	stManualModeParameter[_Chan].stChannelParameter.stManualOption.bTrafoActive := _MachineMode[_Chan].ManualMode.stManualOption.bTrafoActive;
	stManualModeParameter[_Chan].stChannelParameter.stManualOption.bEcsActive := _MachineMode[_Chan].ManualMode.stManualOption.bEcsActive;
	stManualModeParameter[_Chan].stChannelParameter.stManualOption.eZeroOffset := _MachineMode[_Chan].ManualMode.stManualOption.eZeroOffset;					

	_ManualModeJog:=(_MachineMode[_SelectedChannel].ManualMode.nManualTyp=2) AND _Channel[_SelectedChannel].stCmdModesStates.stModes.Manual;
	_ManualModeInc:=(_MachineMode[_SelectedChannel].ManualMode.nManualTyp=3) AND _Channel[_SelectedChannel].stCmdModesStates.stModes.Manual;
	
	stManualModeParameter[_Chan].stAxisParameter.stControlUnit[0].nLogAxisNr := _MachineMode[_Chan].ManualMode.nLogAxisNumber;   (* Log. Achs Nummer *)
	IF stManualModeParameter[_Chan].stAxisParameter.stControlUnit[0].nLogAxisNr = 0 THEN
		stManualModeParameter[_Chan].stAxisParameter.stControlUnit[0].nLogAxisNr := gpCh[_Chan]^.bahn_state.coord_r[0].log_achs_nr_r;
		_MachineMode[_Chan].ManualMode.nLogAxisNumber := gpCh[_Chan]^.bahn_state.coord_r[0].log_achs_nr_r;
	END_IF
	stManualModeParameter[_Chan].stAxisParameter.stControlUnit[0].nSpeed := LREAL_TO_UDINT(_MachineMode[_Chan].ManualMode.nSpeed * (100000/60));//um/min >> mm/sec
	stManualModeControlElements[_Chan].stControlKeys[0].bKeyNeg := _MachineMode[_Chan].ManualMode.bKeyNeg;
	stManualModeControlElements[_Chan].stControlKeys[0].bKeyPos := _MachineMode[_Chan].ManualMode.bKeyPos;
	stManualModeControlElements[_Chan].stControlKeys[0].bKeyRapid := _MachineMode[_Chan].ManualMode.bKeyRapid;
	
	//Handwheel
	IF _Handwheel.xAxisSelect THEN
		_MachineMode[_Chan].ManualMode.nLogAxisNumber := INT_TO_UINT(_Axis[0].nLogAxisNo);
	ELSIF _Handwheel.yAxisSelect THEN
		_MachineMode[_Chan].ManualMode.nLogAxisNumber := INT_TO_UINT(_Axis[1].nLogAxisNo);
	ELSIF _Handwheel.zAxisSelect THEN
		_MachineMode[_Chan].ManualMode.nLogAxisNumber := INT_TO_UINT(_Axis[2].nLogAxisNo);
	ELSIF _Handwheel.aAxisSelect THEN
		_MachineMode[_Chan].ManualMode.nLogAxisNumber := INT_TO_UINT(_Axis[3].nLogAxisNo);
	ELSIF _Handwheel.cAxisSelect THEN
		_MachineMode[_Chan].ManualMode.nLogAxisNumber := INT_TO_UINT(_Axis[4].nLogAxisNo);
	ELSIF _MachineMode[_Chan].ManualMode.nManualTyp = 1 THEN
		_MachineMode[_Chan].ManualMode.nManualTyp := 0;			
	END_IF
	
	IF _Handwheel.x10Resolution THEN
		_MachineMode[_Chan].ManualMode.nHwResolution := 10;
	ELSIF _Handwheel.x100Resolution THEN
		_MachineMode[_Chan].ManualMode.nHwResolution := 100;
	ELSE
		_MachineMode[_Chan].ManualMode.nHwResolution := 1;
	END_IF
		
	stManualModeParameter[_Chan].stChannelParameter.nHandwheelResolution := UDINT_TO_DINT(_MachineMode[_Chan].ManualMode.nHwResolution)* LREAL_TO_DINT(10000);
	_fbUintUdint[_Chan](ninSmall := _Handwheel.Handwheel, nBig := _HandWheelBig);
	stManualModeControlElements[_Chan].nHandwheelinc[0] :=  UDINT_TO_DINT(_HandWheelBig);
	IF _HandWheelBig > 214748364 OR _HandWheelBig = 0 THEN
		_MachineMode[_Chan].ManualMode.nLogAxisNumber := 0;
		_HandWheelBig := 107374182;
	END_IF
END_IF
END_METHOD

METHOD PRIVATE M_Selections
VAR_INPUT
	{attribute 'tc_no_symbol'}
	_Chan					 : INT;
END_VAR
VAR_INST
END_VAR
//Reset
	_MachineMode[_Chan].Reset := Control.Inputs.AlarmAck.Enabled OR Control.Inputs.Reset.Enabled;

//Energize
	_R_Trig[7](CLK:=Energize); 
	IF _R_Trig[7].Q THEN 
		_AutoEn:= TRUE; 
	END_IF
	
	_R_trig[6](CLK:= NOT Energize); 
	IF _R_Trig[6].Q THEN 
		_AutoEn:= FALSE; 
	END_IF

//Stop
	_R_Trig[8](CLK:=Control.PackMLState.Stopping OR Control.PackMLState.Holding);
	_MachineMode[_SelectedChannel].Stop := _R_Trig[8].Q;

//Start
	_R_Trig[9](CLK:= (Control.PackMLState.Starting OR Control.PackMLState.Execute) AND _AxisEnabled);
	_MachineMode[_SelectedChannel].Start := _R_Trig[9].Q;
	
//Standby Mode
	_StandbyMode.Interlock := Control.PackMLState.Execute  OR (_StandbyMode.Enabled AND _MachineMode[_Chan].Mode <> E_CNC_Mode.STANDBY_MODE);
	IF _StandbyMode.Interlock THEN 
		_StandbyMode.Messages := 'CNC Machine Must not be Executing for Standby Mode'; 
	END_IF;
	
	_StandbyMode.Select := (_StandbyMode.Select) AND NOT _StandbyMode.Interlock;
	IF NOT _StandbyMode.Select AND NOT _StandbyMode.Interlock THEN 
		_StandbyMode.Messages := 'CNC Ready for Standby Mode'; 
	END_IF;
	
	_StandbyMode.Queued := _StandbyMode.Select;
	IF _StandbyMode.Queued AND NOT _StandbyMode.Enabled THEN 
		_StandbyMode.Messages := 'CNC Standby Mode Selection Queued'; 
	END_IF;
	
	_R_Trig[10](CLK:= _StandbyMode.Queued); 
	IF _R_Trig[10].Q THEN 
		_MachineMode[_Chan].Standby := TRUE;
	END_IF;
	
	_StandbyMode.Enabled := _StandbyMode.Queued AND _MachineMode[_Chan].Mode = E_CNC_Mode.STANDBY_MODE;
	IF _StandbyMode.Enabled THEN 
		_StandbyMode.Messages := 'CNC Standby Mode Enabled'; 
	END_IF;

//Automatic Mode Selection
	_AutomaticMode.Interlock := Control.PackMLState.Execute AND NOT _AutomaticMode.Enabled OR (_AutomaticMode.Enabled AND _MachineMode[_Chan].Mode <> E_CNC_Mode.AUTOMATIC_MODE);
	IF _AutomaticMode.Interlock THEN 
		_AutomaticMode.Messages := 'CNC Machine Must not be Executing for Automatic Mode Selection'; 
	END_IF;
	
	_AutomaticMode.Select := _AutomaticMode.Select AND NOT _AutomaticMode.Interlock;
	IF NOT _AutomaticMode.Select AND NOT _AutomaticMode.Interlock THEN
 		_AutomaticMode.Messages := 'CNC Ready for Automatic Mode'; 
	END_IF;
	
	_AutomaticMode.Queued := _AutomaticMode.Select;
	IF _AutomaticMode.Queued AND NOT _AutomaticMode.Enabled THEN 
		_AutomaticMode.Messages := 'CNC Automatic Mode Selection Queued'; 
	END_IF;
	
	_R_Trig[11](CLK:= _AutomaticMode.Queued);
	IF _R_Trig[11].Q THEN 
		_MachineMode[_Chan].Automatic := TRUE;
	END_IF;
	
	_AutomaticMode.Enabled := _AutomaticMode.Queued AND _MachineMode[_Chan].Mode = E_CNC_Mode.AUTOMATIC_MODE;
	IF _AutomaticMode.Enabled THEN 
		_AutomaticMode.Messages := 'CNC Automatic Mode Enabled'; 
	END_IF;

//3 MDI Mode Selection
	_MDIMode.Interlock := Control.PackMLState.Execute AND NOT _MDIMode.Enabled  OR (_MDIMode.Enabled AND _MachineMode[_Chan].Mode <> E_CNC_Mode.MDI_MODE);
	IF _MDIMode.Interlock THEN 
		_MDIMode.Messages := 'CNC Machine Must not be Executing for MDI Mode Selection'; 
	END_IF;
	
	_MDIMode.Select := _MDIMode.Select AND NOT _MDIMode.Interlock;
	IF NOT _MDIMode.Select AND NOT _MDIMode.Interlock THEN 
		_MDIMode.Messages := 'CNC Ready for MDI Mode'; 
	END_IF;
	
	_MDIMode.Queued := _MDIMode.Select;
	IF _MDIMode.Queued AND NOT _MDIMode.Enabled THEN 
		_MDIMode.Messages := 'CNC MDI Mode Selection Queued'; 
	END_IF;
	
	_R_Trig[12](CLK:= _MDIMode.Queued); 
	IF _R_Trig[12].Q THEN 
		_MachineMode[_Chan].MDI:= TRUE;
	END_IF;

	_MDIMode.Enabled := _MDIMode.Queued AND _MachineMode[_Chan].Mode = E_CNC_Mode.MDI_MODE;
	IF _MDIMode.Enabled THEN 
		_MDIMode.Messages := 'CNC MDI Mode Enabled'; 
	END_IF;

//Manual Mode Selection
	_ManualMode.Interlock := (NOT control.PackMLState.Stopped AND NOT control.PackMLState.Idle)OR (_ManualMode.Enabled AND ((_MachineMode[_Chan].Mode <> E_CNC_Mode.MANUAL_MODE)OR _R_Trig[15].Q));
	IF _ManualMode.Interlock THEN 
		_ManualMode.Messages := 'CNC Must be in a Stopped or Idle State for Manual Mode'; 
	END_IF;	_R_Trig[13](CLK:= _ManualMode.Queued);
	
	_ManualMode.Select := _ManualMode.Select AND NOT _ManualMode.Interlock;
	IF NOT _ManualMode.Select AND NOT _ManualMode.Interlock THEN 
		_ManualMode.Messages := 'CNC Ready for Manual Mode'; 
	END_IF;
	
	_ManualMode.Queued := _ManualMode.Select;
	IF _ManualMode.Queued AND NOT _ManualMode.Enabled THEN 
		_ManualMode.Messages := 'CNC Manual Mode Selection Queued'; 
	END_IF;

	IF _R_Trig[13].Q THEN 
		_MachineMode[_Chan].ManualMode.nManualTyp := 2;  _MachineMode[_Chan].Manual := TRUE; 
	END_IF;
	
	_ManualMode.Enabled := _ManualMode.Queued AND (_MachineMode[_Chan].ManualMode.nManualTyp<>1) AND _MachineMode[_Chan].Mode = E_CNC_Mode.MANUAL_MODE;
	IF _ManualMode.Enabled THEN 
		_ManualMode.Messages := 'CNC Manual Mode Enabled';
	END_IF;
	
//5 Reference Mode Selection
	_ReferenceMode.Interlock := NOT Control.PackMLState.Resetting OR (_ReferenceMode.Enabled AND _MachineMode[_Chan].Mode <> E_CNC_Mode.REFERENCE_MODE);
	IF _ReferenceMode.Interlock THEN 
		_ReferenceMode.Messages := 'CNC Must be in a Stopped or Resseting State for Reference Mode'; 
	END_IF;
	
	_ReferenceMode.Select := (_ReferenceMode.Select OR _AutoHome OR _ManHome.Enabled) AND NOT _ReferenceMode.Interlock;
	IF NOT _ReferenceMode.Select AND NOT _ReferenceMode.Interlock THEN 
		_ReferenceMode.Messages := 'CNC Ready for Reference Mode'; 
	END_IF;

	_ReferenceMode.Queued := _ReferenceMode.Select;
	IF _ReferenceMode.Queued AND NOT _ReferenceMode.Enabled THEN 
		_ReferenceMode.Messages := 'CNC Reference Mode Selection Queued'; 
	END_IF;

	_ReferenceMode.Enabled := _ReferenceMode.Queued;
	IF _ReferenceMode.Enabled THEN 
		_ReferenceMode.Messages := 'CNC Reference Mode Enabled';
	END_IF;
	
//Handwheel Mode Selected
	_HandwheelMode.Interlock := (NOT control.PackMLState.Stopped AND NOT control.PackMLState.Idle) OR (_HandwheelMode.Enabled AND ((_MachineMode[_Chan].Mode <> E_CNC_Mode.MANUAL_MODE)OR _R_Trig[13].Q));
	IF _HandwheelMode.Interlock THEN 
		_HandwheelMode.Messages := 'CNC Must be in a Stopped or Idle State for Handwheel Mode'; 
	END_IF;

	_HandwheelMode.Select := (_Handwheel.xAxisSelect OR _Handwheel.yAxisSelect OR _Handwheel.zAxisSelect OR _Handwheel.cAxisSelect OR _Handwheel.aAxisSelect) AND NOT _HandwheelMode.Interlock;
	IF NOT _HandwheelMode.Select AND NOT _HandwheelMode.Interlock THEN 
		_HandwheelMode.Messages := 'CNC Ready for Handwheel Mode'; 
	END_IF;

	_HandwheelMode.Queued := _HandwheelMode.Select;
	IF _HandwheelMode.Queued AND NOT _HandwheelMode.Enabled THEN 
		_HandwheelMode.Messages := 'CNC Handwheel Mode Selection Queued'; 
	END_IF;

	_R_Trig[15](CLK:= _HandwheelMode.Queued);
	IF _R_Trig[15].Q THEN 
		_MachineMode[_Chan].ManualMode.nManualTyp := 1; _MachineMode[_Chan].Manual := TRUE; 
	END_IF;

	_HandwheelMode.Enabled := _HandwheelMode.Queued AND (_MachineMode[_Chan].ManualMode.nManualTyp=1) AND _MachineMode[_Chan].Mode = E_CNC_Mode.MANUAL_MODE;
	IF _HandwheelMode.Enabled THEN 
		_HandwheelMode.Messages := 'CNC Handwheel Mode Enabled'; 
	END_IF;

//Manual Home Selection
	_R_Trig[16](CLK:= _Homed);	
	_ManHome.Interlock := (NOT control.PackMLState.Stopped AND NOT control.PackMLState.Resetting) OR _R_Trig[16].Q;
	IF _ManHome.Interlock THEN 
		_ManHome.Messages := 'CNC Must be in a Stopped State for Manual Homing'; 
	END_IF;
	
	_ManHome.Select := _ManHome.Select AND NOT _ManHome.Interlock;
	IF NOT _ManHome.Select AND NOT _ManHome.Interlock THEN 
		_ManHome.Messages := 'CNC Ready for Selected Axis to be Homed'; 
	END_IF;
	
	_ManHome.Queued := _ManHome.Select;
	IF _ManHome.Queued AND NOT _ManHome.Enabled THEN 
		_ManHome.Messages := 'CNC Waiting for Machine to be put into Resetting'; 
	END_IF;
	
	_ManHome.Enabled := _ManHome.Queued AND Control.PackMLState.Resetting;
	IF _ManHome.Enabled THEN 
		_ManHome.Messages := 'CNC Axis Manual Home Enabled'; 
	END_IF;

//Spindle Warmup
	_SpindleWarmup.Interlock := Spindle.Warm OR (NOT A1_Control.PackMLState.Idle AND NOT A1_Control.PackMLState.Starting AND NOT A1_Control.PackMLState.Execute AND NOT A1_Control.PackMLState.Completing);
	IF _SpindleWarmup.Interlock THEN 
		_SpindleWarmup.Messages := 'Spindle is Warm or CNC is Not in a Suitable State'; 
	END_IF;
	
	_SpindleWarmup.Select := _SpindleWarmup.Select AND NOT _SpindleWarmup.Interlock;
	IF NOT _SpindleWarmup.Select AND NOT _SpindleWarmup.Interlock THEN 
		_SpindleWarmup.Messages := 'Ready for Spindle Warmup'; 
	END_IF;
	
	_SpindleWarmup.Queued := _SpindleWarmup.Select;
	IF _SpindleWarmup.Queued AND NOT _SpindleWarmup.Enabled THEN 
		_SpindleWarmup.Messages := 'Spindle Warmup is Queued'; 
	END_IF;
	
	_SpindleWarmup.Enabled := _SpindleWarmup.Queued AND Control.PackMLState.Execute;
	IF _SpindleWarmup.Enabled THEN 
		_SpindleWarmup.Messages := 'Spindle Warmup Enabled'; 
	END_IF;
	
//Retract Tool
	_RetractTool.Interlock := NOT A1_Control.PackMLState.Idle AND NOT A1_Control.PackMLState.Starting AND NOT A1_Control.PackMLState.Execute AND NOT A1_Control.PackMLState.Completing;
	IF _RetractTool.Interlock THEN 
		_RetractTool.Messages := 'Machine Not in a Suitable State to Retract Tool'; 
	END_IF;
	
	_RetractTool.Select := (_RetractTool.Select) AND NOT _RetractTool.Interlock;
	IF NOT _RetractTool.Select AND NOT _RetractTool.Interlock THEN 
		_RetractTool.Messages := 'Ready for Tool Retract'; 
	END_IF;
	
	_RetractTool.Queued := _RetractTool.Select;
	IF _RetractTool.Queued AND NOT _RetractTool.Enabled THEN 
		_RetractTool.Messages := 'Retract Tool Selection Queued'; 
	END_IF;
	
	_RetractTool.Enabled := _RetractTool.Queued AND Control.PackMLState.Execute;
	IF _RetractTool.Enabled THEN 
		_RetractTool.Messages := 'Retract Tool Enabled'; 
	END_IF;
END_METHOD

METHOD PRIVATE M_Spindle
VAR_INPUT
	{attribute 'tc_no_symbol'}
	_Chan					 : INT;
END_VAR
VAR_INST
	_Delay							: TON;
	_fbHandleSpindleTechno			: HLI3_HandleSpindleTechno;
	_ton							: ARRAY[0..5] OF TON;
	_Step							: UINT;
	_MaxSpeed						: UINT := 24000;
	_r_trig							: ARRAY[0..2] OF R_TRIG;
END_VAR
_fbHandleSpindleTechno(
	nHliAxisIdx:=0, 
	nHliChannelIdx:=_Chan, 	
	bIsChannelSpecific:= TRUE,	
	nRevolution=>Spindle.ComVelocity,
	nLogAxisNoChannelSpecific:= 96, 
	nPosition=> Spindle.Position, 
	bError=> Spindle.Error, 
	nErrorId=> Spindle.ErrorID, 
	M03:= Spindle.M3, 
	M04:= Spindle.M4, 
	M05:= Spindle.M5, 
	M19:= Spindle.M19);

Spindle.ActVelocity:= _Axis[5].stStatus.fActVelo;

// Spindle warm up control
_ton[0](PT:=T#90M, IN:= Spindle.Warm AND NOT SC2501.RunFeedback);
IF _ton[0].Q THEN
	Spindle.Warm := FALSE;
END_IF

CASE _Step OF
	0: //Idle
	IF _SpindleWarmup.Queued THEN
		_Step := 1;
	END_IF
	
	1: //Change to MDI Mode
	_r_trig[0](CLK := TRUE);
	IF _r_trig[0].Q THEN
		_MachineMode[_Chan].MDI := TRUE;
	END_IF

	_MachineMode[_Chan].MDIString := 'T6$R$NM06$R$NM03 S12000$R$NG04 120$R$NM03 S18000$R$NG04 120$R$NM03 S24000$R$NG04 60$R$NM05$R$NT0$R$NM06$R$NG84$R$NM30';
	IF _MachineMode[_Chan].Mode = E_CNC_Mode.MDI_MODE THEN
		_r_trig[0](CLK := FALSE);
		_Step := 2;
		
	ELSIF NOT _SpindleWarmup.Queued THEN
		_Step := 0;
		_MachineMode[_Chan].MDIString := '';
		_MachineMode[_Chan].Standby := TRUE;
	END_IF
	
	2: //Start
	Control.Inputs.Start.Enabled:= TRUE;
	
	IF _MachineMode[_Chan].State = E_CNC_State.ACTIVE AND _SpindleWarmup.Enabled THEN
		_r_trig[0](CLK := FALSE);
		_Step := 3;
	ELSIF NOT _SpindleWarmup.Queued THEN
		_Step := 0;
		_MachineMode[_Chan].MDIString := '';
		_MachineMode[_Chan].Standby := TRUE;
	END_IF
	
	3: //Complete
	IF _ProgramEnd[_Chan] THEN
		Spindle.Warm := TRUE;
		_SpindleWarmup.Select:= FALSE;
		_MachineMode[_Chan].MDIString := '';
		_Step := 0;
		_MachineMode[_Chan].Standby := TRUE;
	ELSIF NOT _SpindleWarmup.Enabled THEN
		_Step := 0;
		_MachineMode[_Chan].MDIString := '';
		_MachineMode[_Chan].Standby := TRUE;
	END_IF
END_CASE
END_METHOD

METHOD PRIVATE M_ToolHandler
VAR_INPUT
	{attribute 'tc_no_symbol'}
	_Chan					 : INT;
END_VAR
VAR_INST
	_r_trig					: ARRAY[0..5] OF R_TRIG;
	_f_trig					: ARRAY[0..2] OF F_TRIG;
	_Step					: UINT;
END_VAR
_ToolData[0].tool_desc.tool_id.basic := 0;
_ToolData[0].tool_desc.valid := TRUE;

//Transfer Tool Data for Requested Tool from Database
IF _Channel[_Chan].pChannel^.ToolData.bToolRequest THEN
	CASE _Channel[_Chan].pChannel^.ToolData.nToolRequestID OF
	0:
		_Channel[_Chan].pChannel^.ToolData.stActTool := _ToolData[0];	
	1:
		_Channel[_Chan].pChannel^.ToolData.stActTool := _ToolData[1];	
	2:
		_Channel[_Chan].pChannel^.ToolData.stActTool := _ToolData[2];	
	3:
		_Channel[_Chan].pChannel^.ToolData.stActTool := _ToolData[3];	
	4:
		_Channel[_Chan].pChannel^.ToolData.stActTool := _ToolData[4];	
	5:
		_Channel[_Chan].pChannel^.ToolData.stActTool := _ToolData[5];	
	6:
		_Channel[_Chan].pChannel^.ToolData.stActTool := _ToolData[6];	
		
	END_CASE		
END_IF

//Transfer Tool Data from Currently used tool back into Database
IF _Channel[_Chan].pChannel^.ToolData.bOldToolDataExist THEN
	_Channel[_Chan].pChannel^.ToolData.bOldToolDataExist := FALSE;
END_IF

//Reply of request read and processed
IF _Channel[_Chan].pChannel^.ToolData.nToolRequestID = _Channel[_Chan].pChannel^.ToolData.stActTool.tool_desc.tool_id.basic THEN
	_Channel[_Chan].pChannel^.ToolData.bToolRequest := FALSE;
END_IF

//Tool Holder
_r_trig[0](CLK:= _Channel[_Chan].pChannel^.M[7].bState_rw);
IF _r_trig[0].Q THEN
	Spindle.M7:= TRUE;
END_IF

_f_trig[0](CLK:= Spindle.M7);
IF _f_trig[0].Q THEN
	_Channel[_Chan].pChannel^.M[7].bState_rw:= FALSE;
END_IF

_r_trig[1](CLK:= _Channel[_Chan].pChannel^.M[8].bState_rw);
IF _r_trig[1].Q THEN
	Spindle.M8:= TRUE;
END_IF

_f_trig[1](CLK:= Spindle.M8);
IF _f_trig[1].Q THEN
	_Channel[_Chan].pChannel^.M[8].bState_rw:= FALSE;
END_IF

_r_trig[2](CLK:= _Channel[_Chan].pChannel^.M[9].bState_rw);
IF _r_trig[2].Q THEN
	Spindle.M9:= TRUE;
END_IF

_f_trig[2](CLK:= Spindle.M9);
IF _f_trig[2].Q THEN
	_Channel[_Chan].pChannel^.M[9].bState_rw:= FALSE;
END_IF

//Tool Retract
IF NOT _RetractTool.Queued THEN
	_Step:= 0;
END_IF

CASE _Step OF
	0: //Idle
	IF _RetractTool.Queued THEN
		_Step := 1;
	END_IF
	
	1: //Change to MDI Mode
	_r_trig[3](CLK := TRUE);
	IF _r_trig[3].Q THEN
		_MachineMode[_Chan].MDI := TRUE;
	END_IF
	
	_MachineMode[_Chan].MDIString := 'G85$R$NX8000 Y650 Z-135 C90 A-90$R$NM02';
	IF _MachineMode[_Chan].Mode = E_CNC_Mode.MDI_MODE THEN
		_r_trig[3](CLK := FALSE);
		_Step := 2;
	END_IF
	
	2: //Start
	Control.Inputs.Start.Select:= TRUE;
	
	IF _MachineMode[_Chan].State = E_CNC_State.ACTIVE THEN
		_Step := 3;
	END_IF
	
	3: //Complete
	IF _ProgramEnd[_Chan] THEN//_MachineMode[_Chan].State = E_CNC_State.READY THEN
		_Step := 0;
		_MachineMode[_Chan].MDIString := '';
		_RetractTool.Select:= FALSE;
		_MachineMode[_Chan].Standby := TRUE;
	END_IF
END_CASE
END_METHOD

METHOD PRIVATE M_VariableViewer
VAR_INST
	_fbReadCNCVariables 	: FB_ReadCNCVariables;
END_VAR
_fbReadCNCVariables(
	bEnable:= TRUE, 
	nChanIdx:= _SelectedChannel, 
	eVariablesType:= eVariablesType, 
	tIntervall:= T#1S, 	 
	stCNCVariablesViewer_Data:= stCNCVariablesViewer_Data);

_pVE_Chan0:= HLI3_LinkVEChannelStructure(nChanIdx:= 0, bGlobal:= FALSE);

_pVE_Chan0^.ParkPos.X:=  _ParkPositions[0];
_pVE_Chan0^.ParkPos.Y:=  _ParkPositions[1];
_pVE_Chan0^.ParkPos.Z:=  _ParkPositions[2];
_pVE_Chan0^.ParkPos.C:=  _ParkPositions[3];
_pVE_Chan0^.ParkPos.A:=  _ParkPositions[4];
END_METHOD

METHOD PRIVATE M_WarningMonitor
VAR_INPUT
END_VAR
VAR_INST
END_VAR
VAR_INST // added by the converter: edge detectors and wires of the graphical bodies
    _w1 : BOOL;
END_VAR
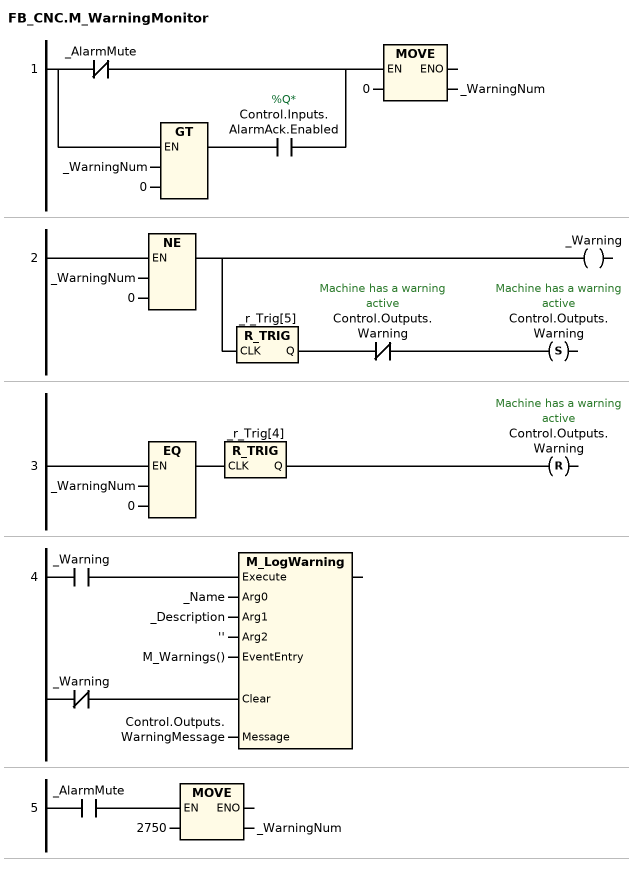
// NETWORK 1
//   Control.Inputs.AlarmAck.Enabled: AT %Q*
IF NOT _AlarmMute OR _WarningNum > 0 AND Control.Inputs.AlarmAck.Enabled THEN _WarningNum := 0; END_IF

// NETWORK 2
//   Control.Outputs.Warning: Machine has a warning active
_w1 := _WarningNum <> 0;
_Warning := _w1;
_r_Trig[5](CLK := _w1); // R_TRIG
Control.Outputs.Warning S= _r_Trig[5].Q AND NOT Control.Outputs.Warning;

// NETWORK 3
//   Control.Outputs.Warning: Machine has a warning active
_r_Trig[4](CLK := _WarningNum = 0); // R_TRIG
Control.Outputs.Warning R= _r_Trig[4].Q;

// NETWORK 4
M_LogWarning(Execute := _Warning, Arg0 := _Name, Arg1 := _Description, Arg2 := '', EventEntry := M_Warnings(), Clear := NOT _Warning, Message := Control.Outputs.WarningMessage);

// NETWORK 5
IF _AlarmMute THEN _WarningNum := 2750; END_IF
END_METHOD

METHOD PRIVATE M_Warnings : TcEventEntry
VAR_INPUT
END_VAR
CASE _WarningNum OF		
	2750: M_Warnings:= TC_Events.TcCnc.W_2750;//Alarm Mute Active						
ELSE
	M_Warnings:=  TC_Events.TcCnc.W_Undefined;
END_CASE
END_METHOD

PROPERTY PUBLIC MachineMode : REFERENCE TO ARRAY[0..3] OF ST_MachineMode;
GET
MachineMode REF= _MachineMode;
END_GET
END_PROPERTY

{attribute 'monitoring' := 'variable'}
PROPERTY PUBLIC Name : String[15]
GET
Name := _Name;
END_GET
SET
_Name := Name;
END_SET
END_PROPERTY

PROPERTY PUBLIC ProgramEnd : REFERENCE TO ARRAY[0..3] OF  BOOL
GET
ProgramEnd REF= _ProgramEnd;
END_GET
END_PROPERTY

PROPERTY PUBLIC ToolData : ARRAY [0..6] OF ST_CNC_TOOL_DATA_EXT
SET
_ToolData:= ToolData;
END_SET
END_PROPERTY

PROPERTY PUBLIC Variables : REFERENCE TO ARRAY[0..9] OF ST_Variable
GET
Variables REF= _Variables;
END_GET
END_PROPERTY

{attribute 'monitoring' := 'variable'}
PROPERTY PUBLIC Warning : Bool
GET
Warning := _Warning;
END_GET
END_PROPERTY

END_FUNCTION_BLOCK

// Objects/FB_CsvLogger_V1_01/FB_CsvLogger
FUNCTION_BLOCK FINAL FB_CsvLogger EXTENDS FB_EventLogger  
VAR_INPUT
	Write					: BOOL;							//Write Log
	HeaderString			: ARRAY[0..9] OF STRING;		//Header Strings
	DataString				: ARRAY[0..9] OF STRING;		//Data Strings
END_VAR                                          	    	
VAR_IN_OUT                                          		
	Control					: ST_System;            		//Machine Control Instance
END_VAR                                             		                                           	
VAR                                                     	
	_Export					: BOOL;							//Export CSV to file destination
	_Fault					: BOOL;	     					//Device Fault
	_SeekPos				: DINT;							//Bytes Logged
	_FaultTimer_ET			: REAL;							//Fault timer elapsed
	_fbCreateDir 			: FB_CreateDir;					//Create File Directory Funciton
	_fbFileOpen				: FB_FileOpen;              	//File Open Function      
	_fbFileClose			: FB_FileClose;             	//File Close Function            
    _fbFileRead             : FB_FileRead;              	//File Read Function 			          
    _fbFileWrite            : FB_FileWrite;             	//File Write Function 	          
	_fbFileDelete  			: FB_FileDelete;            	//File Delete Function           
    _fbFileSeek             : FB_FileSeek;              	//File Seek Function             
	_fbFileTell 			: FB_FileTell;              	//File Tell Function 			          
	_fbFindFileEntry 		: FB_EnumFindFileEntry;     	//File Find File Function 		      
    _hSrcFile               : UINT := 0;					//Temporary file handler
 	_hDestFile              : UINT := 0;					//Export file handler
	_Alarm					: BOOL;							//Device Alarm
	_Warning				: BOOL;							//Device Warning
	_AlarmNum				: DINT;							//Device Alarm Number
	_WarningNum				: DINT;							//Device Warning Number
	_ExtendedErrorCode		: UDINT;						//Extended Error Code
	_R_Trig					: ARRAY[0..9] OF R_TRIG;		//Private Rising Edge Triggers
END_VAR
VAR PERSISTENT
	_Enable					: BOOL;							//Enable CSV logging
	_MaxFileSize			: DINT := 100000;           	//Maximum file size in bytes
	_Name					: STRING[15];					//Name for HMI
	_Description			: STRING[40];					//Description for HMI
	_AlarmMute				: BOOL;							//Alarm Mute
	_FaultTimer_PT			: REAL;							//Fault timer preset time
	_TempFilePath			: STRING:='C:\TwinCAT\3.1\Boot\';//Temporary File Path
	_ExportFilePath			: STRING:='C:\TwinCAT\';		//Export File Path
END_VAR

M_AlarmMonitor();
M_WarningMonitor();
M_Log();

{attribute 'monitoring' := 'variable'}
PROPERTY PUBLIC Alarm : Bool
GET
Alarm := _Alarm;
END_GET
END_PROPERTY

{attribute 'monitoring' := 'variable'}
PROPERTY PUBLIC AlarmMute : BOOL
SET
AlarmMute := _AlarmMute;
END_SET
END_PROPERTY

{attribute 'monitoring' := 'variable'}
PROPERTY PUBLIC Description : String[40]
GET
Description := _Description;
END_GET
SET
_Description := Description;
END_SET
END_PROPERTY

{attribute 'monitoring' := 'variable'}
PROPERTY PUBLIC Enable : BOOL
GET
Enable := _Enable;
END_GET
SET
_Enable := Enable;
END_SET
END_PROPERTY

{attribute 'monitoring' := 'variable'}
PROPERTY PUBLIC Fault : Bool
SET
_Fault := Fault;
END_SET
END_PROPERTY

{attribute 'monitoring' := 'variable'}
PROPERTY PUBLIC FaultTimer_ET : real
GET
FaultTimer_ET := _FaultTimer_ET;
END_GET
END_PROPERTY

{attribute 'monitoring' := 'variable'}
PROPERTY PUBLIC FaultTimer_PT : real
GET
FaultTimer_PT := _FaultTimer_PT;
END_GET
SET
_FaultTimer_PT := FaultTimer_PT;
END_SET
END_PROPERTY

METHOD FB_exit : BOOL
VAR_INPUT
	bInCopyCode : BOOL; // if TRUE, the exit method is called for exiting an instance that is copied afterwards (online change).
END_VAR
IF _hSrcFile <> 0 THEN
	_fbFileClose( bExecute := FALSE );	
	_fbFileClose(sNetId:='', hFile:=_hSrcFile, bExecute:=TRUE, tTimeout:=DEFAULT_ADS_TIMEOUT);
END_IF
END_METHOD

METHOD PRIVATE M_AlarmMonitor
VAR_INPUT
END_VAR
VAR_INST // added by the converter: edge detectors and wires of the graphical bodies
    _w1, _w2, _w3, _w4, _w5, _w6, _w7 : BOOL;
    _rt1, _rt2, _rt3, _rt4, _rt5, _rt6, _rt7, _rt8, _rt9, _rt10 : R_TRIG;
END_VAR
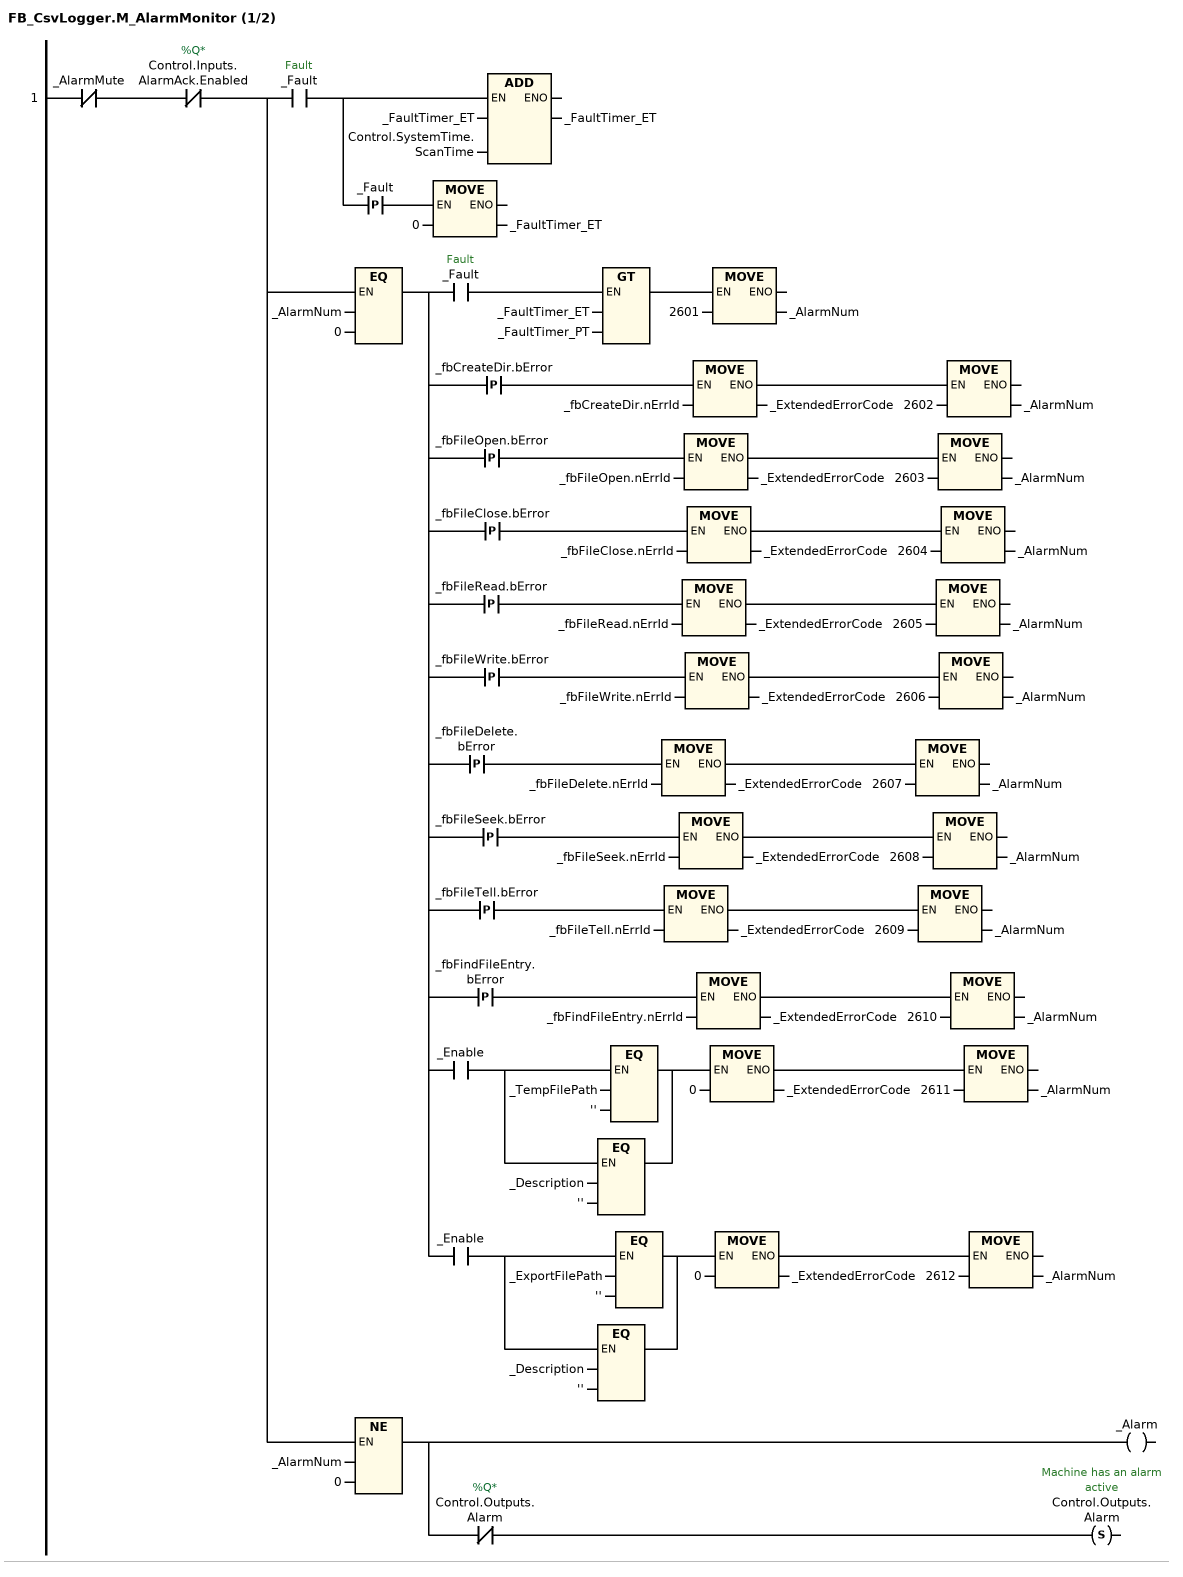
// NETWORK 1
//   Control.Inputs.AlarmAck.Enabled: AT %Q*
//   _Fault: Fault
//   _FaultTimer_ET: Fault timer elapsed
//   Control.SystemTime.ScanTime: Last scan time (Seconds)
//   _FaultTimer_PT: Fault timer preset time
//   Control.Outputs.Alarm: AT %Q* | Machine has an alarm active
_w1 := NOT _AlarmMute AND NOT Control.Inputs.AlarmAck.Enabled;
_w2 := _w1 AND _Fault;
IF _w2 THEN _FaultTimer_ET := _FaultTimer_ET + Control.SystemTime.ScanTime; END_IF
_rt1(CLK := _Fault);
IF _w2 AND _rt1.Q THEN _FaultTimer_ET := 0; END_IF
_w3 := _w1 AND _AlarmNum = 0;
IF _w3 AND _Fault AND _FaultTimer_ET > _FaultTimer_PT THEN _AlarmNum := 2601; END_IF
_rt2(CLK := _fbCreateDir.bError);
IF _w3 AND _rt2.Q THEN _ExtendedErrorCode := _fbCreateDir.nErrId; END_IF
IF _w3 AND _rt2.Q THEN _AlarmNum := 2602; END_IF
_rt3(CLK := _fbFileOpen.bError);
IF _w3 AND _rt3.Q THEN _ExtendedErrorCode := _fbFileOpen.nErrId; END_IF
IF _w3 AND _rt3.Q THEN _AlarmNum := 2603; END_IF
_rt4(CLK := _fbFileClose.bError);
IF _w3 AND _rt4.Q THEN _ExtendedErrorCode := _fbFileClose.nErrId; END_IF
IF _w3 AND _rt4.Q THEN _AlarmNum := 2604; END_IF
_rt5(CLK := _fbFileRead.bError);
IF _w3 AND _rt5.Q THEN _ExtendedErrorCode := _fbFileRead.nErrId; END_IF
IF _w3 AND _rt5.Q THEN _AlarmNum := 2605; END_IF
_rt6(CLK := _fbFileWrite.bError);
IF _w3 AND _rt6.Q THEN _ExtendedErrorCode := _fbFileWrite.nErrId; END_IF
IF _w3 AND _rt6.Q THEN _AlarmNum := 2606; END_IF
_rt7(CLK := _fbFileDelete.bError);
IF _w3 AND _rt7.Q THEN _ExtendedErrorCode := _fbFileDelete.nErrId; END_IF
IF _w3 AND _rt7.Q THEN _AlarmNum := 2607; END_IF
_rt8(CLK := _fbFileSeek.bError);
IF _w3 AND _rt8.Q THEN _ExtendedErrorCode := _fbFileSeek.nErrId; END_IF
IF _w3 AND _rt8.Q THEN _AlarmNum := 2608; END_IF
_rt9(CLK := _fbFileTell.bError);
IF _w3 AND _rt9.Q THEN _ExtendedErrorCode := _fbFileTell.nErrId; END_IF
IF _w3 AND _rt9.Q THEN _AlarmNum := 2609; END_IF
_rt10(CLK := _fbFindFileEntry.bError);
IF _w3 AND _rt10.Q THEN _ExtendedErrorCode := _fbFindFileEntry.nErrId; END_IF
IF _w3 AND _rt10.Q THEN _AlarmNum := 2610; END_IF
_w4 := _w3 AND _Enable;
IF _w4 AND _TempFilePath = '' OR _w4 AND _Description = '' THEN _ExtendedErrorCode := 0; END_IF
IF _w4 AND _TempFilePath = '' OR _w4 AND _Description = '' THEN _AlarmNum := 2611; END_IF
_w5 := _w3 AND _Enable;
IF _w5 AND _ExportFilePath = '' OR _w5 AND _Description = '' THEN _ExtendedErrorCode := 0; END_IF
IF _w5 AND _ExportFilePath = '' OR _w5 AND _Description = '' THEN _AlarmNum := 2612; END_IF
_w6 := _w1 AND _AlarmNum <> 0;
_Alarm := _w6;
Control.Outputs.Alarm S= _w6 AND NOT Control.Outputs.Alarm;

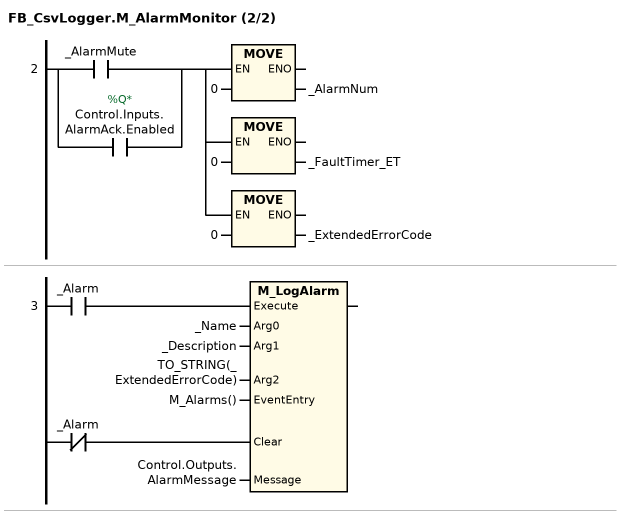
// NETWORK 2
//   Control.Inputs.AlarmAck.Enabled: AT %Q*
//   _FaultTimer_ET: Fault timer elapsed
//   _ExtendedErrorCode: Fault timer elapsed
_w7 := _AlarmMute OR Control.Inputs.AlarmAck.Enabled;
IF _w7 THEN _AlarmNum := 0; END_IF
IF _w7 THEN _FaultTimer_ET := 0; END_IF
IF _w7 THEN _ExtendedErrorCode := 0; END_IF

// NETWORK 3
M_LogAlarm(Execute := _Alarm, Arg0 := _Name, Arg1 := _Description, Arg2 := TO_STRING(_ExtendedErrorCode), EventEntry := M_Alarms(), Clear := NOT _Alarm, Message := Control.Outputs.AlarmMessage);
END_METHOD

METHOD PRIVATE M_Alarms : TcEventEntry
VAR_INPUT
END_VAR
CASE _AlarmNum OF
	2601: M_Alarms:= TC_Events.TcCsvLogger.A_2601;//Alarm
	2602: M_Alarms:= TC_Events.TcCsvLogger.A_2602;//Create File Directory Error 
	2603: M_Alarms:= TC_Events.TcCsvLogger.A_2603;//File Open Error
	2604: M_Alarms:= TC_Events.TcCsvLogger.A_2604;//File Close Error
	2605: M_Alarms:= TC_Events.TcCsvLogger.A_2605;//File Read Error			
	2606: M_Alarms:= TC_Events.TcCsvLogger.A_2606;//File Write Error		
	2607: M_Alarms:= TC_Events.TcCsvLogger.A_2607;//File Delete Error	
	2608: M_Alarms:= TC_Events.TcCsvLogger.A_2608;//File Seek Error
	2609: M_Alarms:= TC_Events.TcCsvLogger.A_2609;//File Tell Error			
	2610: M_Alarms:= TC_Events.TcCsvLogger.A_2610;//File Find File Error		
	2611: M_Alarms:= TC_Events.TcCsvLogger.A_2611;//Temporary File Path or Name Error		
	2612: M_Alarms:= TC_Events.TcCsvLogger.A_2612;//Export File Path or Name Error				
ELSE
	M_Alarms:= TC_Events.TcCsvLogger.A_Undefined;
END_CASE
END_METHOD

METHOD PUBLIC M_Log
VAR_INST
	{attribute 'tc_no_symbol'}
	_Step								: UINT;
	{attribute 'tc_no_symbol'}
	_Timeout							: TON;
	{attribute 'tc_no_symbol'}
    _buffRead                			: ARRAY[1..100000] OF BYTE;
	{attribute 'tc_no_symbol'}
 	_cbReadLength            			: UDINT := 0;
	{attribute 'tc_no_symbol'}
	_HeaderString						: T_MAXSTRING;
	{attribute 'tc_no_symbol'}
	_DataString							: T_MAXSTRING;
	{attribute 'tc_no_symbol'}
	_TimeStamp							: STRING(31);
	{attribute 'tc_no_symbol'}
	_Value								: INT;
END_VAR
CASE _Step OF
	0:  // Step 0: Wait for open file request
		IF _Enable AND NOT _Alarm THEN
			_Step := 1; 
		END_IF
	1:  // Step 1: Check if temporary directory exists	
		_fbFindFileEntry(bExecute:= FALSE);
		_fbFindFileEntry(sPathName:= LEFT(_TempFilePath,LEN(_TempFilePath)-1), eCmd:= eEnumCmd_First, bExecute:= TRUE, tTimeout:= DEFAULT_ADS_TIMEOUT);
		IF _fbFindFileEntry.bBusy THEN _Step := 2; END_IF
	2:  // Step 2: Wait for temporary directory check	
		_fbFindFileEntry( bExecute := FALSE );
		IF NOT _fbFindFileEntry.bBusy AND NOT _fbFindFileEntry.bError THEN 
			IF _fbFindFileEntry.stFindFile.fileAttributes.bDirectory THEN
				_Step := 5; 
			ELSE
				_Step := 3; 
			END_IF
		END_IF
	3:  // Step 3: Create temporary directory
	    _hSrcFile:=0;
		_fbCreateDir( bExecute := FALSE );
		_fbCreateDir(sNetId:= '', sPathName := _TempFilePath, ePath:= PATH_GENERIC, bExecute:= TRUE, tTimeout:= DEFAULT_ADS_TIMEOUT);
		IF _fbCreateDir.bBusy THEN _Step := 4; END_IF
	4:  // Step 4: Wait for temporary directory to be created
		_fbCreateDir( bExecute := FALSE );
		IF NOT _fbCreateDir.bBusy AND NOT _fbCreateDir.bError THEN _Step := 5; END_IF
	5:  // Step 5: Check if temporary file exists	
		_fbFindFileEntry(bExecute:= FALSE);
		_fbFindFileEntry(sPathName:= concat(_TempFilePath,concat(_Description,'.csv')), eCmd:= eEnumCmd_First, bExecute:= TRUE, tTimeout:= DEFAULT_ADS_TIMEOUT);
		IF _fbFindFileEntry.bBusy THEN _Step := 6; END_IF
	6:  // Step 6: Wait for temporary file check	
		_fbFindFileEntry( bExecute := FALSE );
		IF NOT _fbFindFileEntry.bBusy AND NOT _fbFindFileEntry.bError THEN 
			IF _fbFindFileEntry.stFindFile.fileAttributes.bArchive THEN
				_fbFileOpen.nMode := FOPEN_MODEREAD OR FOPEN_MODEPLUS;
			ELSE
				_fbFileOpen.nMode := FOPEN_MODEWRITE; 
			END_IF
			_Step := 7; 
		END_IF	
	7:  // Step 7: Open temporary CSV file
		_fbFileOpen( bExecute := FALSE );
		_fbFileOpen( sNetId := '', sPathName := concat(_TempFilePath,concat(_Description,'.csv')), ePath := PATH_GENERIC, tTimeout := DEFAULT_ADS_TIMEOUT, bExecute := TRUE );
		IF _fbFileOpen.bBusy THEN _Step := 8; END_IF
	8:	// Step 8: Wait for temporary CSV to be created
		_fbFileOpen( bExecute := FALSE, hFile=> _hSrcFile);
		IF NOT _fbFileOpen.bBusy AND NOT _fbFileOpen.bError THEN 
			IF _fbFileOpen.nMode = (FOPEN_MODEREAD OR FOPEN_MODEPLUS) THEN
				_Step := 9; 
			ELSE
				_Step := 11; 
			END_IF
		END_IF	
	9:  // Step 9: Find if header exists 
        _fbFileRead( bExecute:= FALSE );
        _fbFileRead( sNetId:='', hFile:=_hSrcFile, bExecute:=TRUE, pReadBuff:= ADR(_buffRead), cbReadLen:= SIZEOF(_buffRead), tTimeout:=DEFAULT_ADS_TIMEOUT);
        _Step := 10;
    10:  // Step 10: Wait for feedback of header existance
        _fbFileRead( bExecute:= FALSE );
        IF NOT _fbFileRead.bBusy AND NOT _fbFileRead.bError THEN
			IF _fbFileRead.cbReadLen > 0 THEN // Header already exists
				_Step := 13; 
			ELSE
				_Step := 11; 
			END_IF
        END_IF
	11:	// Step 11: Write header string to temporary CSV file
		_fbFileWrite( bExecute := FALSE);
		_HeaderString := '';
		FOR _Value:= 0 TO UINT_TO_INT(SIZEOF(HeaderString)/SIZEOF(STRING))-1 BY 1 DO
			IF _Value < UINT_TO_INT((SIZEOF(HeaderString)/SIZEOF(STRING))-1) THEN
				IF HeaderString[_Value+1] <> '' THEN
			    	_HeaderString := concat(_HeaderString,concat(HeaderString[_Value],','));	
				ELSE
					_HeaderString := concat(_HeaderString,concat(HeaderString[_Value],'$0D'));
					EXIT;
				END_IF
			ELSE
				_HeaderString := concat(_HeaderString,concat(HeaderString[_Value],'$0D'));
			END_IF 
		END_FOR;
		_fbFileWrite( sNetId:='', hFile:= _hSrcFile, pWriteBuff:= ADR(_HeaderString), cbWriteLen:= INT_TO_UINT(Len(_HeaderString)), bExecute:=TRUE, tTimeout:=DEFAULT_ADS_TIMEOUT);
		IF _fbFileWrite.bBusy THEN _Step := 12; END_IF
	12:	// Step 12: Wait for CSV header to be written
		_fbFileWrite( bExecute := FALSE );
		IF NOT _fbFileWrite.bBusy AND NOT _fbFileWrite.bError THEN 
			_Step := 13; 
		END_IF	
	13:	// Step 13: Get the current position of the file pointer
		_fbFileTell(bExecute:= FALSE);
		_fbFileTell(hFile:= _hSrcFile, bExecute:= TRUE);
		IF _fbFileTell.bBusy THEN _Step := 14; END_IF
	14:	// Step 14: Wait for file tell
		_fbFileTell(bExecute:= FALSE, nSeekPos => _SeekPos);
		IF NOT _fbFileTell.bBusy AND NOT _fbFileTell.bError THEN 
			_Step := 15; 
		END_IF	
	15:	// Step 15: Set the current position of the file pointer
		_fbFileSeek(bExecute:= FALSE);
		_fbFileSeek(eOrigin:= SEEK_SET, nSeekPos:= _SeekPos + 1, hFile:= _hSrcFile, bExecute:= TRUE);
		IF _fbFileSeek.bBusy THEN _Step := 16; END_IF
	16:	// Step 16: Wait for file seek
		_fbFileSeek(bExecute:= FALSE);
		IF NOT _fbFileSeek.bBusy AND NOT _fbFileSeek.bError THEN 
			_Step := 17; 
		END_IF	
	17: // Step 17: Wait for write or export request
		_R_Trig[0](CLK:= _Export);
		_R_Trig[1](CLK:= Write);
		IF _R_Trig[0].Q THEN
			_Step := 22;
		ELSIF _R_Trig[1].Q THEN
 			_Step := 18;
		ELSIF NOT _Enable THEN
			_Step := 36;
		END_IF
	18:	// Step 18: Write data to CSV file
		_fbFileWrite( bExecute := FALSE);
		_DataString := '';
		FOR _Value:= 0 TO UINT_TO_INT(SIZEOF(DataString)/SIZEOF(STRING))-1 BY 1 DO
			IF _Value < UINT_TO_INT((SIZEOF(DataString)/SIZEOF(STRING))-1) THEN
				IF DataString[_Value+1] <> '' THEN
			    	_DataString := concat(_DataString,concat(DataString[_Value],','));	
				ELSE
					_DataString := concat(_DataString,concat(DataString[_Value],'$0D'));
					EXIT;
				END_IF
			ELSE
				_DataString := concat(_DataString,concat(DataString[_Value],'$0D'));
			END_IF 
		END_FOR;
		_fbFileWrite( sNetId:='', hFile:= _hSrcFile, pWriteBuff:= ADR(_DataString), cbWriteLen:= INT_TO_UINT(Len(_DataString)), bExecute:=TRUE, tTimeout:=T#3S );
		IF _fbFileWrite.bBusy THEN _Step := 19; END_IF
	19:	// Step 19: Wait for CSV data to be written
		_fbFileWrite( bExecute := FALSE );
		IF NOT _fbFileWrite.bBusy AND NOT _fbFileWrite.bError THEN 
			_Step := 20; 
		END_IF		
	20:	// Step 20: Get the current position of the file pointer
		_fbFileTell(bExecute:= FALSE);
		_fbFileTell(hFile:= _hSrcFile, bExecute:= TRUE);
		IF _fbFileTell.bBusy THEN _Step := 21; END_IF
	21:	// Step 21: Wait for file tell
		_fbFileTell(bExecute:= FALSE, nSeekPos => _SeekPos);
		IF NOT _fbFileTell.bBusy AND NOT _fbFileTell.bError THEN 
			IF (_SeekPos > _MaxFileSize) OR (DINT_TO_UDINT(_SeekPos) > SIZEOF(_buffRead)) THEN
				_SeekPos := LEN(_HeaderString);
				_Step := 15; 
			ELSE 
				_Step := 17; 
			END_IF
		END_IF	
	22: // Step 22: Close temporary CSV 
		IF _hSrcFile <> 0 THEN
			_fbFileClose( bExecute := FALSE );	
			_fbFileClose(sNetId:='', hFile:=_hSrcFile, bExecute:=TRUE, tTimeout:=DEFAULT_ADS_TIMEOUT);
			IF _fbFileClose.bBusy THEN _Step := 23; END_IF
		ELSE
			_Step := 24;
		END_IF
	23:	// Step 23: Wait for temporary CSV to close
		_fbFileClose( bExecute := FALSE );
		IF NOT _fbFileClose.bBusy AND NOT _fbFileClose.bError THEN 
			_hSrcFile := 0;
			_Step := 24;
		END_IF
	24: // Step 24: Open temporary CSV file
		_fbFileOpen( bExecute := FALSE );
		_fbFileOpen( sNetId := '', sPathName := concat(_TempFilePath,concat(_Description,'.csv')),nMode := FOPEN_MODEREAD, ePath := PATH_GENERIC, tTimeout := DEFAULT_ADS_TIMEOUT, bExecute := TRUE );
		IF _fbFileOpen.bBusy THEN _Step := 25; END_IF
	25:	// Step 25: Wait for temporary CSV to be created
		_fbFileOpen( bExecute := FALSE, hFile=> _hSrcFile);
		IF NOT _fbFileOpen.bBusy AND NOT _fbFileOpen.bError THEN _Step := 26; END_IF	
	26: // Step 26: Check if export directory exists	
		_fbFindFileEntry(bExecute:= FALSE);
		_fbFindFileEntry(sPathName:= LEFT(_ExportFilePath,LEN(_ExportFilePath)-1), eCmd:= eEnumCmd_First, bExecute:= TRUE, tTimeout:= DEFAULT_ADS_TIMEOUT);
		IF _fbFindFileEntry.bBusy THEN _Step := 27; END_IF
	27: // Step 27: Wait for export directory check	
		_fbFindFileEntry( bExecute := FALSE );
		IF NOT _fbFindFileEntry.bBusy AND NOT _fbFindFileEntry.bError THEN 
			IF _fbFindFileEntry.stFindFile.fileAttributes.bDirectory THEN
				_Step := 30; 
			ELSE
				_Step := 28; 
			END_IF
		END_IF
	28: // Step 28: Create export directory
        _hDestFile:=0;
		_fbCreateDir( bExecute := FALSE );
		_fbCreateDir(sNetId:= '', sPathName := _ExportFilePath, ePath:= PATH_GENERIC, bExecute:= TRUE, tTimeout:= DEFAULT_ADS_TIMEOUT);
		IF _fbCreateDir.bBusy AND NOT _fbCreateDir.bError THEN _Step := 29; END_IF
	29: // Step 29: Wait for export directory to be created
		_fbCreateDir( bExecute := FALSE );
		IF NOT _fbCreateDir.bBusy THEN _Step := 30; END_IF
	30: // Step 30: Create export CSV file
		_fbFileOpen( bExecute := FALSE );
		_timeStamp := concat(LEFT(SystemTime_To_String(Control.SystemTime.CurrentTime),10),concat(' ',concat(TO_STRING(Control.SystemTime.CurrentTime.wHour),concat('-',concat(TO_STRING(Control.SystemTime.CurrentTime.wMinute),concat('-',TO_STRING(Control.SystemTime.CurrentTime.wSecond)))))));
		_fbFileOpen( sNetId := '', sPathName := concat(_ExportFilePath,concat(_TimeStamp,concat(' ',concat(_Description,'.csv')))),nMode := FOPEN_MODEAPPEND, ePath := PATH_GENERIC, tTimeout := DEFAULT_ADS_TIMEOUT, bExecute := TRUE );
		IF _fbFileOpen.bBusy THEN _Step := 31; END_IF
	31:	// Step 31: Wait for export CSV to be created
		_fbFileOpen( bExecute := FALSE, hFile=> _hDestFile);
		IF NOT _fbFileOpen.bBusy AND NOT _fbFileOpen.bError THEN _Step := 32; END_IF	
    32: // Step 32: Read data from temporary file 
        _cbReadLength := 0;
        _fbFileRead( bExecute:= FALSE );
        _fbFileRead( sNetId:='', hFile:=_hSrcFile , pReadBuff:= ADR(_buffRead), cbReadLen:= SIZEOF(_buffRead),bExecute:=TRUE, tTimeout:=T#60S);
        _Step := 33;
    33:	// Step 33: Wait for temporary file to be read
        _fbFileRead( bExecute:= FALSE );
        IF NOT _fbFileRead.bBusy AND NOT _fbFileRead.bError THEN
        	_cbReadLength := _fbFileRead.cbRead;
            _Step := 34;
        END_IF
    34: // Step 34: Write data to export file 
        _fbFileWrite( bExecute := FALSE );
        _fbFileWrite( sNetId:='', hFile:=_hDestFile,pWriteBuff:= ADR(_buffRead), cbWriteLen:= _cbReadLength, bExecute:=TRUE, tTimeout:=T#60S);
        _Step := 35;
    35: // Step 35: Wait for export file to be written
       	_fbFileWrite( bExecute := FALSE );
        IF NOT _fbFileWrite.bBusy THEN
             IF _fbFileWrite.bError THEN
                  _Step := 42;
             ELSE
             	IF _fbFileRead.bEOF THEN//Check if the EOF flag ist set 
                   _Step := 36;//Cleanup: close the export and temporary files 
               	ELSE
                   _Step := 32;//Repeat reading/writing 
               	END_IF
            END_IF
        END_IF
	36: // Step 36: Close export CSV file
		IF _hDestFile <> 0 THEN
			_fbFileClose( bExecute := FALSE );	
			_fbFileClose(sNetId:='', hFile:=_hDestFile, bExecute:=TRUE, tTimeout:=DEFAULT_ADS_TIMEOUT);
			IF _fbFileClose.bBusy THEN _Step := 37; END_IF
		ELSE
			_Step := 38;
		END_IF
	37:	// Step 37: Wait for export CSV to close
		_fbFileClose( bExecute := FALSE );
		IF NOT _fbFileClose.bBusy AND NOT _fbFileClose.bError THEN 
			_hDestFile := 0;
			_Step := 38;
		END_IF
	38: // Step 38: Close temporary CSV file
		IF _hSrcFile <> 0 THEN
			_fbFileClose( bExecute := FALSE );	
			_fbFileClose(sNetId:='', hFile:=_hSrcFile, bExecute:=TRUE, tTimeout:=DEFAULT_ADS_TIMEOUT);
			IF _fbFileClose.bBusy THEN _Step := 39; END_IF
		ELSE
			_Step := 42;
		END_IF
	39:	// Step 39: Wait for temporary CSV to close
		_fbFileClose( bExecute := FALSE );
		IF NOT _fbFileClose.bBusy AND NOT _fbFileClose.bError THEN 
			_hSrcFile := 0;
			_Step := 40;
		END_IF
	40:  // Step 40: Delete temporary CSV file
		_fbFileDelete( bExecute := FALSE );	
		_fbFileDelete(sNetId:='', sPathName:= concat(_TempFilePath,concat(_Description,'.csv')), ePath:= PATH_GENERIC, bExecute:=TRUE, tTimeout:=DEFAULT_ADS_TIMEOUT);
		IF _fbFileDelete.bBusy THEN _Step := 41; END_IF
	41:	// Step 33: Wait for temporary CSV to Delete
		_fbFileDelete( bExecute := FALSE );
		IF NOT _fbFileDelete.bBusy AND NOT _fbFileDelete.bError THEN 
			_Step := 42;
		END_IF
    42: // Step 42: Cleanup 
        IF _hDestFile <> 0 THEN
        	_Step := 36;//Close the export file
        ELSIF _hSrcFile <> 0 THEN
        	_Step := 38;//Close and delete the temporary file 
        ELSE
        	_Step := 0;
        END_IF	
	
END_CASE

// Error Handling
_Timeout(In:=_Step > 0 AND _Step <> 17 ,PT:=T#60S);
_R_Trig[6](clk:= _Timeout.Q OR _Alarm);
IF _R_Trig[6].Q THEN _STEP := 36; END_IF
END_METHOD

METHOD PRIVATE M_WarningMonitor
VAR_INPUT
END_VAR
VAR_INST
END_VAR
VAR_INST // added by the converter: edge detectors and wires of the graphical bodies
    _w1 : BOOL;
END_VAR
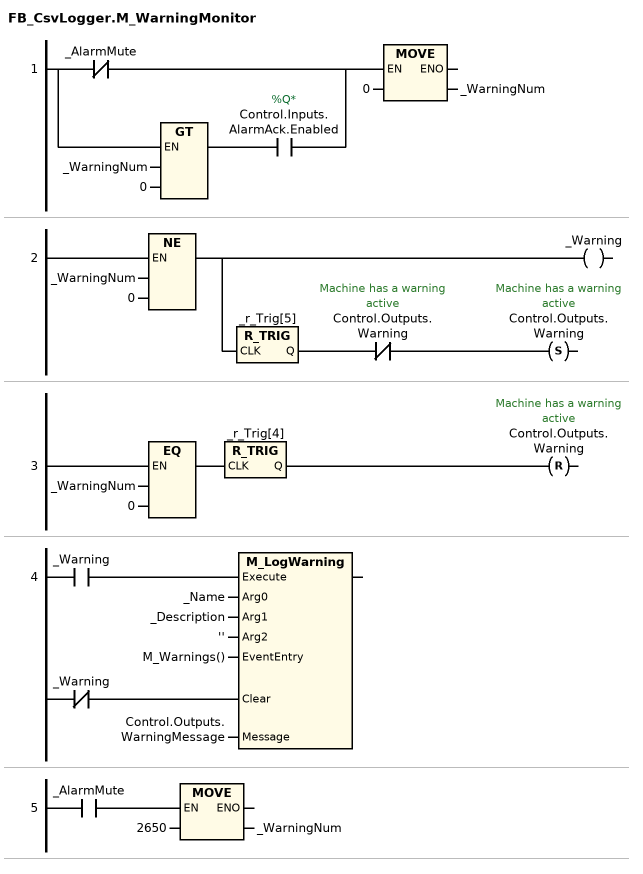
// NETWORK 1
//   Control.Inputs.AlarmAck.Enabled: AT %Q*
IF NOT _AlarmMute OR _WarningNum > 0 AND Control.Inputs.AlarmAck.Enabled THEN _WarningNum := 0; END_IF

// NETWORK 2
//   Control.Outputs.Warning: Machine has a warning active
_w1 := _WarningNum <> 0;
_Warning := _w1;
_r_Trig[5](CLK := _w1); // R_TRIG
Control.Outputs.Warning S= _r_Trig[5].Q AND NOT Control.Outputs.Warning;

// NETWORK 3
//   Control.Outputs.Warning: Machine has a warning active
_r_Trig[4](CLK := _WarningNum = 0); // R_TRIG
Control.Outputs.Warning R= _r_Trig[4].Q;

// NETWORK 4
M_LogWarning(Execute := _Warning, Arg0 := _Name, Arg1 := _Description, Arg2 := '', EventEntry := M_Warnings(), Clear := NOT _Warning, Message := Control.Outputs.WarningMessage);

// NETWORK 5
IF _AlarmMute THEN _WarningNum := 2650; END_IF
END_METHOD

METHOD PRIVATE M_Warnings : TcEventEntry
VAR_INPUT
END_VAR
CASE _WarningNum OF
	2650: M_Warnings:= TC_Events.TcCsvLogger.W_2650;//Alarm Mute							
ELSE
	M_Warnings:=  TC_Events.TcCsvLogger.W_Undefined;
END_CASE
END_METHOD

{attribute 'monitoring' := 'variable'}
PROPERTY PUBLIC Name : String[15]
GET
Name := _Name;
END_GET
SET
_Name := Name;
END_SET
END_PROPERTY

{attribute 'monitoring' := 'variable'}
PROPERTY PUBLIC Warning : Bool
GET
Warning := _Warning;
END_GET
END_PROPERTY

END_FUNCTION_BLOCK

// Objects/FB_Cylinder_V4_01/FB_Cylinder
FUNCTION_BLOCK FINAL FB_Cylinder EXTENDS FB_EventLogger 
VAR_INPUT
	Energized						: BOOL;							//Optional Energize Input
END_VAR                                                     		
VAR_IN_OUT                                                  		
	Control							: ST_System;					//Machine Control Instance
END_VAR                                                     		
VAR                                                         		
	_AutoExtend						: BOOL;							//Automated Extend Signal
	_AutoRetract					: BOOL;							//Automated Retract Signal
	_ManExtend						: BOOL;							//Screen Selection
	_ManRetract						: BOOL;							//Screen Selection
	_ManOff							: BOOL;							//Screen Selection
	_ForceExtend					: BOOL;							//Screen Selection
	_ForceRetract					: BOOL;							//Screen Selection
	_ForceOff						: BOOL;							//Screen Selection
	_CycleEnable					: BOOL;							//Cylinder Cylce Enable
	_ExtendReed1		AT %I*		: BOOL;							//Cylinder Extend Reed 1
	_ExtendReed2		AT %I*		: BOOL;							//Cylinder Extend Reed 2
	_ExtendReed3		AT %I*		: BOOL;							//Cylinder Extend Reed 3
	_ExtendReed4		AT %I*		: BOOL;							//Cylinder Extend Reed 4
	_RetractReed1		AT %I*		: BOOL;							//Cylinder Retract Reed 1
	_RetractReed2		AT %I*		: BOOL;							//Cylinder Retract Reed 2
	_RetractReed3		AT %I*		: BOOL;							//Cylinder Retract Reed 3
	_RetractReed4		AT %I*		: BOOL;							//Cylinder Retract Reed 4
	_DualSolenoid					: BOOL;							//Configured as a dual Solenoid Device
	_SingleSolenoidNormal			: BOOL;							//Configured as a Signal Solenoid Extend Device (Default)	
	_SingleSolenoidReverse			: BOOL;							//Configured as a Signal Solenoid Retract Device
	_CountsReset					: BOOL;							//Cycle Counts Reset
	_CycleExtend					: BOOL;							//Cylinder Cycle Extend
	_CycleRetract					: BOOL;							//Cylinder Cycle Retract
	_ExtendSolOnTime_ET				: REAL;							//Time Extend Solenoid Has Been Energised
	_ExtendSolOffTime_ET			: REAL;							//Time Since Extend Solenoid was Last Energised
	_RetractSolOnTime_ET			: REAL;							//Time Retract Solenoid Has Been Energised
	_RetractSolOffTime_ET			: REAL;							//Time Since Retract Solenoid was Last Energised
	_ExtendTime_ET					: REAL;							//Time Cylinder has been Extended
	_RetractTime_ET					: REAL;							//Time Cylinder has been Retracted
	_CycleExtTime_ET				: REAL;							//Cylinder Cycle Extend Accumulated Time
	_CycleRetTime_ET				: REAL;							//Cylinder Cycle Retract Accumulated Time
	_ExtendReed						: BOOL;							//All cylinder extend reeds have been made
	_RetractReed					: BOOL;							//All cylinder retract reeds have been made
	_ReedFaultCount					: SINT;							//Count for type of reed fault
	_ExtendSol				AT %Q*	: BOOL;							//Physical output for extend solenoid
	_RetractSol				AT %Q*	: BOOL;							//Physical output for retract solenoid
	_ExtendFault					: BOOL;							//Fault for cylinder extend
	_RetractFault					: BOOL;							//Fault for cylinder retract
	_ReedFault						: BOOL;							//Fault for reed
	_ReedFaultTime_ET				: REAL;							//Reed fault elapsed time
	_ExFaultTime_ET					: REAL;							//Extend fault elapsed time
	_RtFaultTime_ET					: REAL;							//Retract fault elapsed time
	_Alarm							: BOOL;							//Device Alarm
	_Warning						: BOOL;							//Device Warning
	_AlarmNum						: DINT;							//Device Alarm Number
	_WarningNum						: DINT;							//Device Warning Number
	_Mute_Retract					: BOOL;							//Mute Retract Alarm
	_Mute_Extend					: BOOL;							//Mute Extend Alarm
	_extendReedUsed1				: BOOL;                 	
	_extendReedUsed2				: BOOL;                 	
	_extendReedUsed3				: BOOL;                 	
	_extendReedUsed4				: BOOL;                 	
	_retractReedUsed1				: BOOL;
	_retractReedUsed2				: BOOL;
	_retractReedUsed3				: BOOL;
	_retractReedUsed4				: BOOL;
	_R_Trig							: ARRAY[0..19] OF R_TRIG;		//Private Rising Edge Triggers
END_VAR
VAR PERSISTENT
	_Name							: STRING[15];					//Name for HMI
	_Description					: STRING[40];					//Description for HMI
	_AlarmMute						: BOOL;							//Alarm Mute
	_TypeCfg						: E_CylinderTypeConfig;			//Type Selection from Screen
	_ExtendReedsUsed				: WORD;							//Data Word for Number of Extend Reeds used
	_RetractReedsUsed				: WORD;							//Data Word for Number of Retract Reeds used
	_ExtendCount					: REAL;							//Total number of cylinder extends
	_RetractCount					: REAL;							//Total number of cylinder retracts
	_ReedFaultTime_PT				: REAL;							//Reed Fault Preset Time
	_ExFaultTime_PT					: REAL;							//Extend Fault Preset Time
	_RtFaultTime_PT					: REAL;							//Retract Fault Preset Time
	_CycleExtTime_PT				: REAL;							//Cylinder Cycle Extend Time Preset
	_CycleRetTime_PT				: REAL;							//Cylinder Cycle Retract Time Preset
	_Variables						: ARRAY [0..9] OF ST_Variable;	//Device Associated Varibles Array	
END_VAR

M_AlarmMonitor();
M_WarningMonitor();
M_CountsReset();
M_UnlatchManuals();
M_TypeConfig();
M_TestCycle();
M_Extend();
M_Retract();
M_ExtendFault();
M_RetractFault();
M_ReedFault();
M_ReedControl();

{attribute 'monitoring' := 'variable'}
PROPERTY PUBLIC Alarm : Bool
GET
Alarm := _Alarm;
END_GET
END_PROPERTY

{attribute 'monitoring' := 'variable'}
PROPERTY PUBLIC AlarmMute : BOOL
SET
AlarmMute := _AlarmMute;
END_SET
END_PROPERTY

{attribute 'monitoring' := 'variable'}
PROPERTY PUBLIC AutoExtend : Bool
SET
_AutoExtend:= AutoExtend;
END_SET
END_PROPERTY

{attribute 'monitoring' := 'variable'}
PROPERTY PUBLIC AutoRetract : Bool
SET
_AutoRetract:= AutoRetract;
END_SET
END_PROPERTY

{attribute 'monitoring' := 'variable'}
PROPERTY PUBLIC CycleExtTime_PT : real
GET
CycleExtTime_PT := _CycleExtTime_PT;
END_GET
SET
_CycleExtTime_PT := CycleExtTime_PT;
END_SET
END_PROPERTY

{attribute 'monitoring' := 'variable'}
PROPERTY PUBLIC CycleRetTime_PT : real
GET
CycleRetTime_PT := _CycleRetTime_PT;
END_GET
SET
_CycleRetTime_PT := CycleRetTime_PT;
END_SET
END_PROPERTY

{attribute 'monitoring' := 'variable'}
PROPERTY PUBLIC Description : String[40]
GET
Description := _Description;
END_GET
SET
_Description := Description;
END_SET
END_PROPERTY

{attribute 'monitoring' := 'variable'}
PROPERTY PUBLIC ExFaultTime_ET : real
GET
ExFaultTime_ET := _ExFaultTime_ET;
END_GET
END_PROPERTY

{attribute 'monitoring' := 'variable'}
PROPERTY PUBLIC ExFaultTime_PT : real
GET
ExFaultTime_PT := _ExFaultTime_PT;
END_GET
SET
_ExFaultTime_PT := ExFaultTime_PT;
END_SET
END_PROPERTY

{attribute 'monitoring' := 'variable'}
PROPERTY PUBLIC ExtendReed : Bool
GET
ExtendReed := _ExtendReed;
END_GET
END_PROPERTY

{attribute 'monitoring' := 'variable'}
PROPERTY PUBLIC ExtendReed1 : Bool
GET
ExtendReed1 := _ExtendReed;
END_GET
SET
PUBLIC 
VAR
END_VAR
_ExtendReed1 := ExtendReed1;
END_SET
END_PROPERTY

{attribute 'monitoring' := 'variable'}
PROPERTY PUBLIC ExtendSol : Bool
GET
ExtendSol := _ExtendSol;
END_GET
END_PROPERTY

{attribute 'monitoring' := 'variable'}
PROPERTY PUBLIC ForceExtend : Bool
GET
ForceExtend := _ForceExtend;
END_GET
SET
_ForceExtend := ForceExtend;
END_SET
END_PROPERTY

{attribute 'monitoring' := 'variable'}
PROPERTY PUBLIC ForceRetract : Bool
GET
ForceRetract := _ForceRetract;
END_GET
SET
_ForceRetract := ForceRetract;
END_SET
END_PROPERTY

METHOD PRIVATE M_AlarmMonitor
VAR_INPUT
END_VAR
VAR_INST // added by the converter: edge detectors and wires of the graphical bodies
    _w1, _w2, _w3, _w4, _w5 : BOOL;
END_VAR
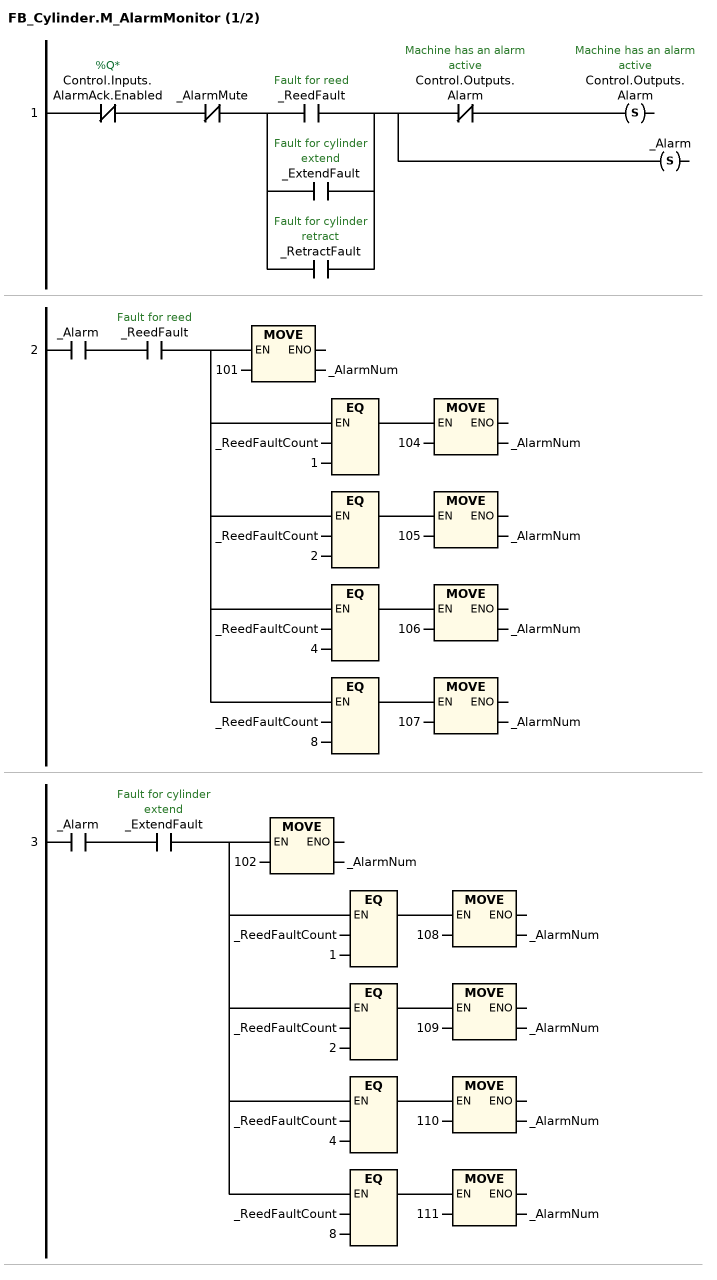
// NETWORK 1
//   Control.Inputs.AlarmAck.Enabled: AT %Q*
//   _ReedFault: Fault for reed
//   _ExtendFault: Fault for cylinder extend
//   _RetractFault: Fault for cylinder retract
//   Control.Outputs.Alarm: Machine has an alarm active
_w1 := NOT Control.Inputs.AlarmAck.Enabled AND NOT _AlarmMute AND (_ReedFault OR _ExtendFault OR _RetractFault);
Control.Outputs.Alarm S= _w1 AND NOT Control.Outputs.Alarm;
_Alarm S= _w1;

// NETWORK 2
//   _ReedFault: Fault for reed
//   _ReedFaultCount: Count for type of reed fault
_w2 := _Alarm AND _ReedFault;
IF _w2 THEN _AlarmNum := 101; END_IF
IF _w2 AND _ReedFaultCount = 1 THEN _AlarmNum := 104; END_IF
IF _w2 AND _ReedFaultCount = 2 THEN _AlarmNum := 105; END_IF
IF _w2 AND _ReedFaultCount = 4 THEN _AlarmNum := 106; END_IF
IF _w2 AND _ReedFaultCount = 8 THEN _AlarmNum := 107; END_IF

// NETWORK 3
//   _ExtendFault: Fault for cylinder extend
//   _ReedFaultCount: Count for type of reed fault
_w3 := _Alarm AND _ExtendFault;
IF _w3 THEN _AlarmNum := 102; END_IF
IF _w3 AND _ReedFaultCount = 1 THEN _AlarmNum := 108; END_IF
IF _w3 AND _ReedFaultCount = 2 THEN _AlarmNum := 109; END_IF
IF _w3 AND _ReedFaultCount = 4 THEN _AlarmNum := 110; END_IF
IF _w3 AND _ReedFaultCount = 8 THEN _AlarmNum := 111; END_IF

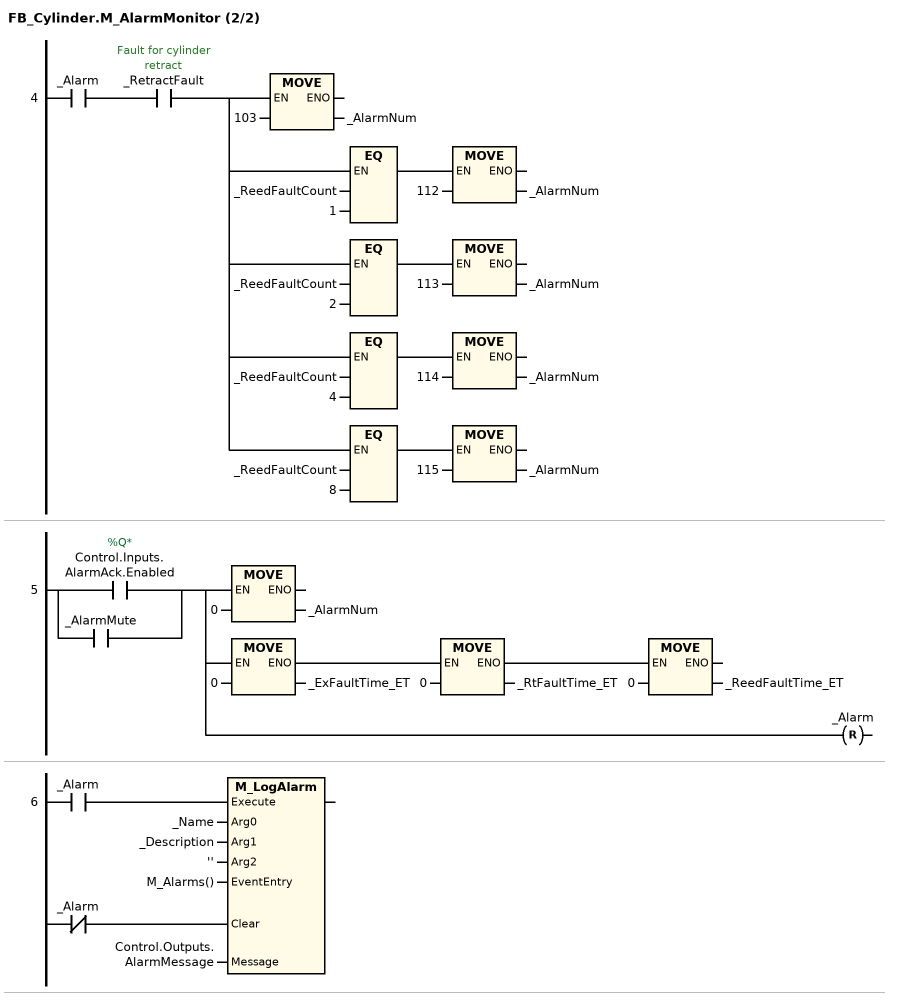
// NETWORK 4
//   _RetractFault: Fault for cylinder retract
//   _ReedFaultCount: Count for type of reed fault
_w4 := _Alarm AND _RetractFault;
IF _w4 THEN _AlarmNum := 103; END_IF
IF _w4 AND _ReedFaultCount = 1 THEN _AlarmNum := 112; END_IF
IF _w4 AND _ReedFaultCount = 2 THEN _AlarmNum := 113; END_IF
IF _w4 AND _ReedFaultCount = 4 THEN _AlarmNum := 114; END_IF
IF _w4 AND _ReedFaultCount = 8 THEN _AlarmNum := 115; END_IF

// NETWORK 5
//   Control.Inputs.AlarmAck.Enabled: AT %Q*
//   _ExFaultTime_ET: Extend fault elapsed time
//   _RtFaultTime_ET: Retract fault elapsed time
//   _ReedFaultTime_ET: Reed fault elapsed time
_w5 := Control.Inputs.AlarmAck.Enabled OR _AlarmMute;
IF _w5 THEN _AlarmNum := 0; END_IF
IF _w5 THEN _ExFaultTime_ET := 0; END_IF
IF _w5 THEN _RtFaultTime_ET := 0; END_IF
IF _w5 THEN _ReedFaultTime_ET := 0; END_IF
_Alarm R= _w5;

// NETWORK 6
M_LogAlarm(Execute := _Alarm, Arg0 := _Name, Arg1 := _Description, Arg2 := '', EventEntry := M_Alarms(), Clear := NOT _Alarm, Message := Control.Outputs.AlarmMessage);
END_METHOD

METHOD PRIVATE M_Alarms : TcEventEntry
VAR_INPUT
END_VAR
CASE _AlarmNum OF
	101: M_Alarms:= TC_Events.TcCylinder.A_101;//Reed Alarm
	102: M_Alarms:= TC_Events.TcCylinder.A_102;//Extend Alarm	
	103: M_Alarms:= TC_Events.TcCylinder.A_103;//Retract Alarm
	104: M_Alarms:= TC_Events.TcCylinder.A_104;//Reed A Alarm
	105: M_Alarms:= TC_Events.TcCylinder.A_105;//Reed B Alarm		
	106: M_Alarms:= TC_Events.TcCylinder.A_106;//Reed C Alarm		
	107: M_Alarms:= TC_Events.TcCylinder.A_107;//Reed D Alarm
	108: M_Alarms:= TC_Events.TcCylinder.A_108;//Extend Reed A Alarm
	109: M_Alarms:= TC_Events.TcCylinder.A_109;//Extend Reed B Alarm
	110: M_Alarms:= TC_Events.TcCylinder.A_110;//Extend Reed C Alarm	
	111: M_Alarms:= TC_Events.TcCylinder.A_111;//Extend Reed D Alarm		
	112: M_Alarms:= TC_Events.TcCylinder.A_112;//Retract Reed A Alarm	
	113: M_Alarms:= TC_Events.TcCylinder.A_113;//Retract Reed B Alarm	
	114: M_Alarms:= TC_Events.TcCylinder.A_114;//Retract Reed C Alarm
	115: M_Alarms:= TC_Events.TcCylinder.A_115;//Retract Reed D Alarm
ELSE
	M_Alarms:= TC_Events.TcCylinder.A_Undefined;
END_CASE
END_METHOD

METHOD PRIVATE M_CountsReset
VAR_INPUT
END_VAR
IF _CountsReset THEN
	_ExtendCount := 0;
	_RetractCount := 0;
END_IF
END_METHOD

METHOD PRIVATE M_Extend
VAR_INPUT
END_VAR
VAR_INST // added by the converter: edge detectors and wires of the graphical bodies
    _w1, _w2 : BOOL;
END_VAR
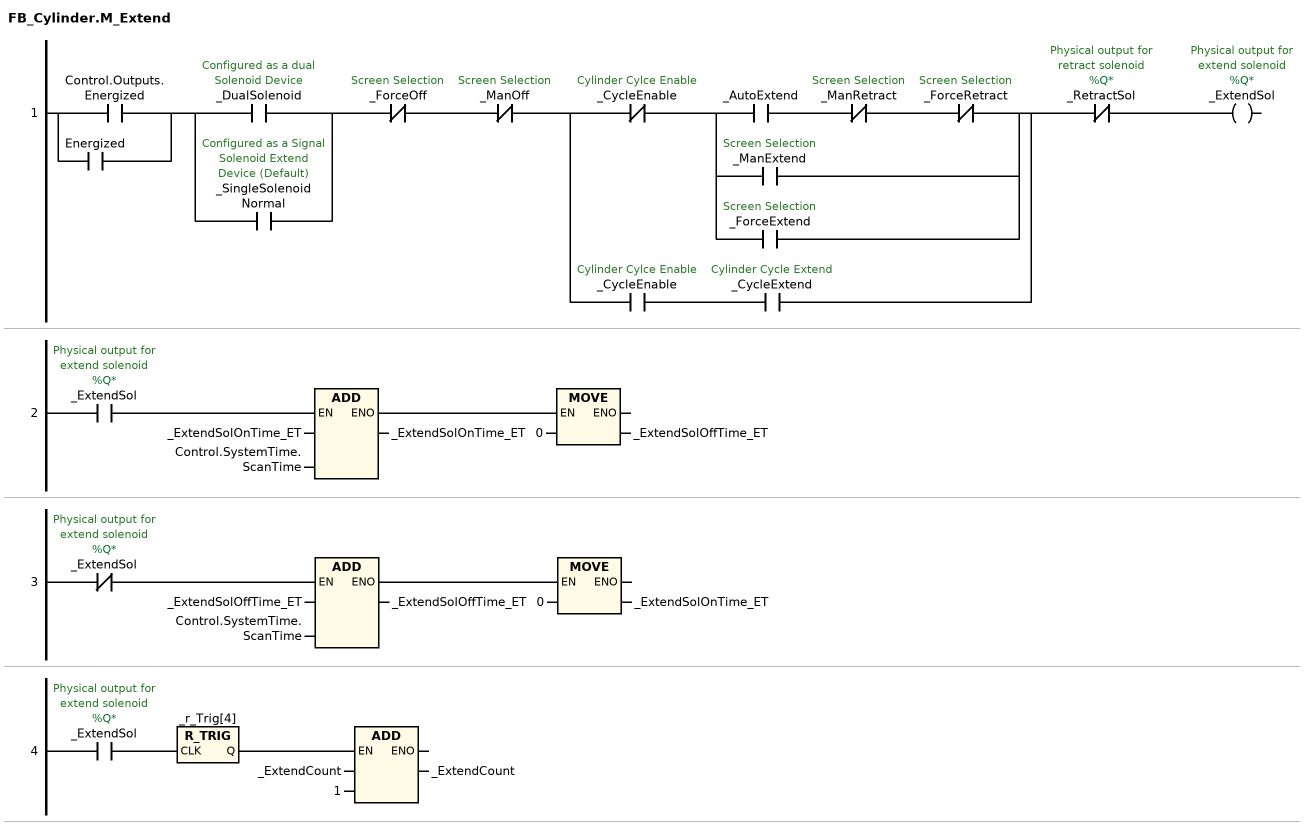
// NETWORK 1
//   _DualSolenoid: Configured as a dual Solenoid Device
//   _SingleSolenoidNormal: Configured as a Signal Solenoid Extend Device (Default)
//   _ForceOff: Screen Selection
//   _ManOff: Screen Selection
//   _CycleEnable: Cylinder Cylce Enable
//   _ManRetract: Screen Selection
//   _ForceRetract: Screen Selection
//   _ManExtend: Screen Selection
//   _ForceExtend: Screen Selection
//   _CycleExtend: Cylinder Cycle Extend
//   _RetractSol: Physical output for retract solenoid | AT %Q*
//   _ExtendSol: Physical output for extend solenoid | AT %Q*
_ExtendSol := (Control.Outputs.Energized OR Energized) AND (_DualSolenoid OR _SingleSolenoidNormal) AND NOT _ForceOff AND NOT _ManOff AND (NOT _CycleEnable AND (_AutoExtend AND NOT _ManRetract AND NOT _ForceRetract OR _ManExtend OR _ForceExtend) OR _CycleEnable AND _CycleExtend) AND NOT _RetractSol;

// NETWORK 2
//   _ExtendSol: Physical output for extend solenoid | AT %Q*
//   _ExtendSolOnTime_ET: Time Extend Solenoid Has Been Energised
//   Control.SystemTime.ScanTime: Last scan time (Seconds)
//   _ExtendSolOffTime_ET: Time Since Extend Solenoid was Last Energised
_w1 := _ExtendSol;
IF _w1 THEN _ExtendSolOnTime_ET := _ExtendSolOnTime_ET + Control.SystemTime.ScanTime; END_IF
IF _w1 THEN _ExtendSolOffTime_ET := 0; END_IF

// NETWORK 3
//   _ExtendSol: Physical output for extend solenoid | AT %Q*
//   _ExtendSolOffTime_ET: Time Since Extend Solenoid was Last Energised
//   Control.SystemTime.ScanTime: Last scan time (Seconds)
//   _ExtendSolOnTime_ET: Time Extend Solenoid Has Been Energised
_w2 := NOT _ExtendSol;
IF _w2 THEN _ExtendSolOffTime_ET := _ExtendSolOffTime_ET + Control.SystemTime.ScanTime; END_IF
IF _w2 THEN _ExtendSolOnTime_ET := 0; END_IF

// NETWORK 4
//   _ExtendSol: Physical output for extend solenoid | AT %Q*
//   _ExtendCount: Total number of cylinder extends
_r_Trig[4](CLK := _ExtendSol); // R_TRIG
IF _r_Trig[4].Q THEN _ExtendCount := _ExtendCount + 1; END_IF
END_METHOD

METHOD PRIVATE M_ExtendFault
VAR_INPUT
END_VAR
VAR_INST
	_extending					: BOOL;
	_extendReedFault_Q			: BOOL;
	_extendReedFaultArray		: ARRAY[0..4] OF BOOL;
END_VAR
VAR_INST // added by the converter: edge detectors and wires of the graphical bodies
    _w1, _w2, _w3, _w4, _w5 : BOOL;
END_VAR
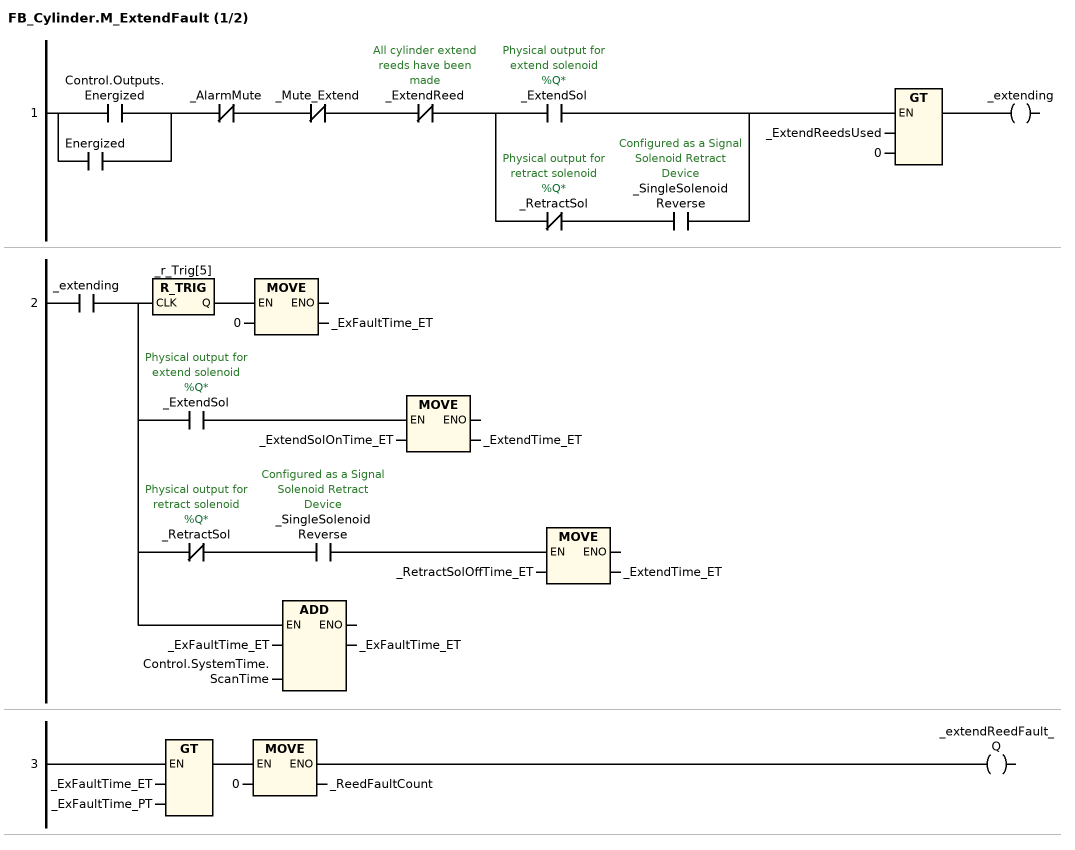
// NETWORK 1
//   _ExtendReed: All cylinder extend reeds have been made
//   _ExtendSol: Physical output for extend solenoid | AT %Q*
//   _RetractSol: Physical output for retract solenoid | AT %Q*
//   _SingleSolenoidReverse: Configured as a Signal Solenoid Retract Device
//   _ExtendReedsUsed: Data Word for Number of Extend Reeds used
_extending := (Control.Outputs.Energized OR Energized) AND NOT _AlarmMute AND NOT _Mute_Extend AND NOT _ExtendReed AND (_ExtendSol OR NOT _RetractSol AND _SingleSolenoidReverse) AND _ExtendReedsUsed > 0;

// NETWORK 2
//   _ExFaultTime_ET: Extend fault elapsed time
//   _ExtendSol: Physical output for extend solenoid | AT %Q*
//   _ExtendSolOnTime_ET: Time Extend Solenoid Has Been Energised
//   _ExtendTime_ET: Time Cylinder has been Extended
//   _RetractSol: Physical output for retract solenoid | AT %Q*
//   _SingleSolenoidReverse: Configured as a Signal Solenoid Retract Device
//   _RetractSolOffTime_ET: Time Since Retract Solenoid was Last Energised
//   Control.SystemTime.ScanTime: Last scan time (Seconds)
_r_Trig[5](CLK := _extending); // R_TRIG
IF _r_Trig[5].Q THEN _ExFaultTime_ET := 0; END_IF
IF _extending AND _ExtendSol THEN _ExtendTime_ET := _ExtendSolOnTime_ET; END_IF
IF _extending AND NOT _RetractSol AND _SingleSolenoidReverse THEN _ExtendTime_ET := _RetractSolOffTime_ET; END_IF
IF _extending THEN _ExFaultTime_ET := _ExFaultTime_ET + Control.SystemTime.ScanTime; END_IF

// NETWORK 3
//   _ExFaultTime_ET: Extend fault elapsed time
//   _ReedFaultCount: Count for type of reed fault
_w1 := _ExFaultTime_ET > _ExFaultTime_PT;
IF _w1 THEN _ReedFaultCount := 0; END_IF
_extendReedFault_Q := _w1;

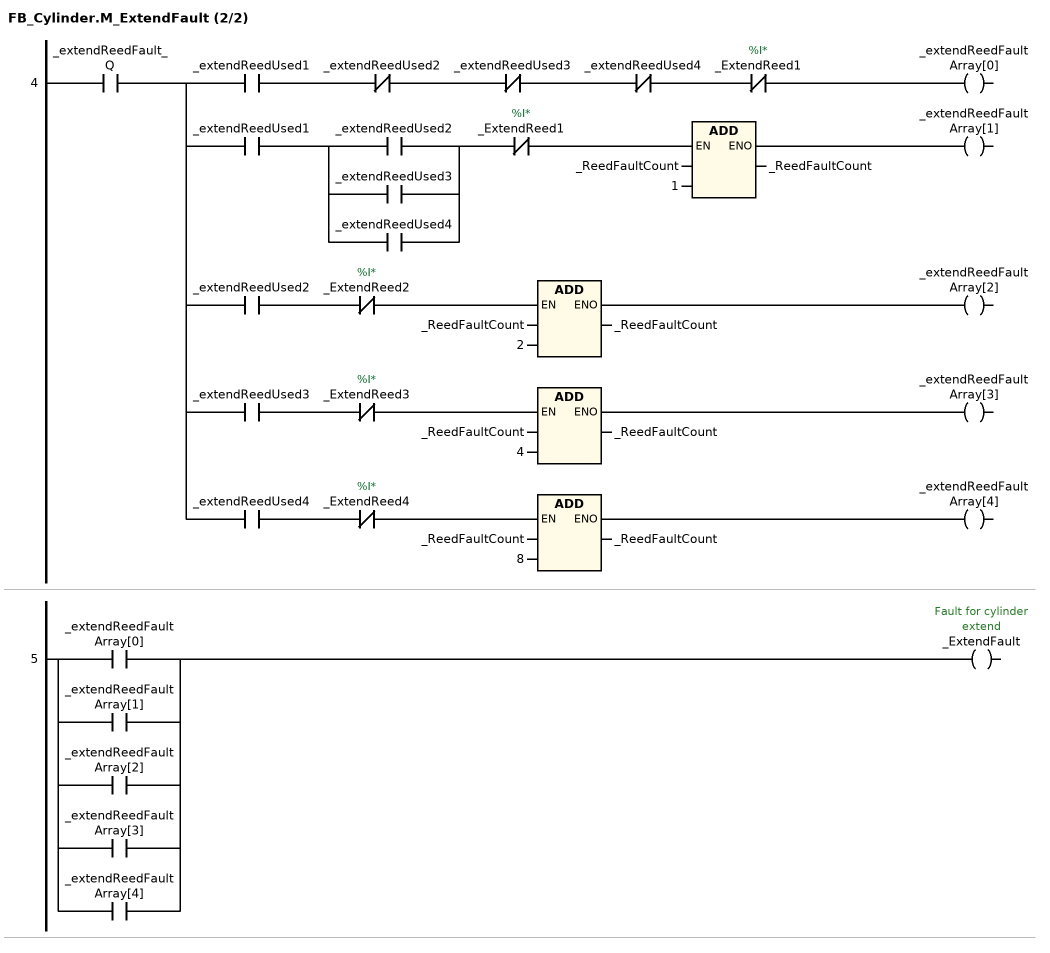
// NETWORK 4
//   _ExtendReed1: AT %I*
//   _ReedFaultCount: Count for type of reed fault
//   _ExtendReed2: AT %I*
//   _ExtendReed3: AT %I*
//   _ExtendReed4: AT %I*
_extendReedFaultArray[0] := _extendReedFault_Q AND _extendReedUsed1 AND NOT _extendReedUsed2 AND NOT _extendReedUsed3 AND NOT _extendReedUsed4 AND NOT _ExtendReed1;
_w2 := _extendReedFault_Q AND _extendReedUsed1 AND (_extendReedUsed2 OR _extendReedUsed3 OR _extendReedUsed4) AND NOT _ExtendReed1;
IF _w2 THEN _ReedFaultCount := _ReedFaultCount + 1; END_IF
_extendReedFaultArray[1] := _w2;
_w3 := _extendReedFault_Q AND _extendReedUsed2 AND NOT _ExtendReed2;
IF _w3 THEN _ReedFaultCount := _ReedFaultCount + 2; END_IF
_extendReedFaultArray[2] := _w3;
_w4 := _extendReedFault_Q AND _extendReedUsed3 AND NOT _ExtendReed3;
IF _w4 THEN _ReedFaultCount := _ReedFaultCount + 4; END_IF
_extendReedFaultArray[3] := _w4;
_w5 := _extendReedFault_Q AND _extendReedUsed4 AND NOT _ExtendReed4;
IF _w5 THEN _ReedFaultCount := _ReedFaultCount + 8; END_IF
_extendReedFaultArray[4] := _w5;

// NETWORK 5
//   _ExtendFault: Fault for cylinder extend
_ExtendFault := _extendReedFaultArray[0] OR _extendReedFaultArray[1] OR _extendReedFaultArray[2] OR _extendReedFaultArray[3] OR _extendReedFaultArray[4];
END_METHOD

METHOD PRIVATE M_ReedControl
VAR_INPUT
END_VAR
VAR_INST
END_VAR
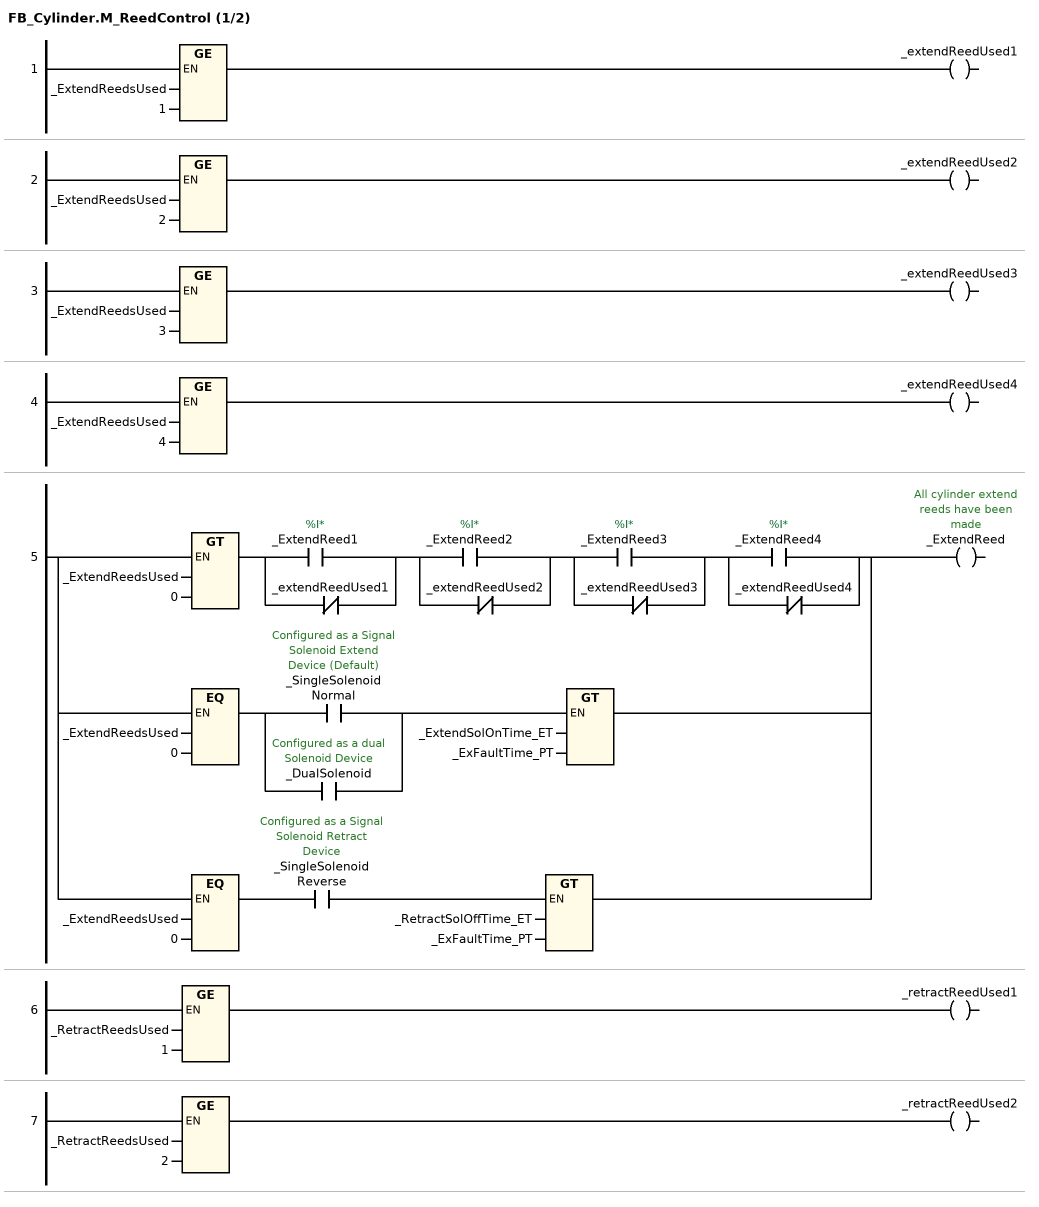
// NETWORK 1
//   _ExtendReedsUsed: Data Word for Number of Extend Reeds used
_extendReedUsed1 := _ExtendReedsUsed >= 1;

// NETWORK 2
//   _ExtendReedsUsed: Data Word for Number of Extend Reeds used
_extendReedUsed2 := _ExtendReedsUsed >= 2;

// NETWORK 3
//   _ExtendReedsUsed: Data Word for Number of Extend Reeds used
_extendReedUsed3 := _ExtendReedsUsed >= 3;

// NETWORK 4
//   _ExtendReedsUsed: Data Word for Number of Extend Reeds used
_extendReedUsed4 := _ExtendReedsUsed >= 4;

// NETWORK 5
//   _ExtendReedsUsed: Data Word for Number of Extend Reeds used
//   _ExtendReed1: AT %I*
//   _ExtendReed2: AT %I*
//   _ExtendReed3: AT %I*
//   _ExtendReed4: AT %I*
//   _SingleSolenoidNormal: Configured as a Signal Solenoid Extend Device (Default)
//   _DualSolenoid: Configured as a dual Solenoid Device
//   _ExtendSolOnTime_ET: Time Extend Solenoid Has Been Energised
//   _SingleSolenoidReverse: Configured as a Signal Solenoid Retract Device
//   _RetractSolOffTime_ET: Time Since Retract Solenoid was Last Energised
//   _ExtendReed: All cylinder extend reeds have been made
_ExtendReed := _ExtendReedsUsed > 0 AND (_ExtendReed1 OR NOT _extendReedUsed1) AND (_ExtendReed2 OR NOT _extendReedUsed2) AND (_ExtendReed3 OR NOT _extendReedUsed3) AND (_ExtendReed4 OR NOT _extendReedUsed4) OR _ExtendReedsUsed = 0 AND (_SingleSolenoidNormal OR _DualSolenoid) AND _ExtendSolOnTime_ET > _ExFaultTime_PT OR _ExtendReedsUsed = 0 AND _SingleSolenoidReverse AND _RetractSolOffTime_ET > _ExFaultTime_PT;

// NETWORK 6
//   _RetractReedsUsed: Data Word for Number of Retract Reeds used
_retractReedUsed1 := _RetractReedsUsed >= 1;

// NETWORK 7
//   _RetractReedsUsed: Data Word for Number of Retract Reeds used
_retractReedUsed2 := _RetractReedsUsed >= 2;

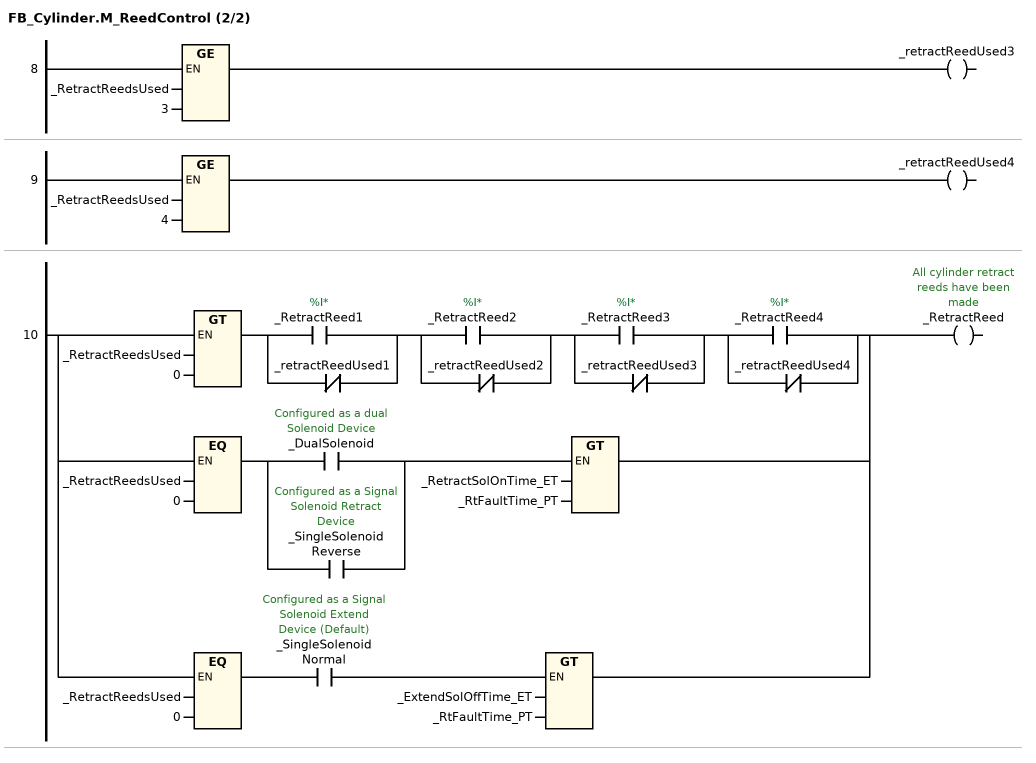
// NETWORK 8
//   _RetractReedsUsed: Data Word for Number of Retract Reeds used
_retractReedUsed3 := _RetractReedsUsed >= 3;

// NETWORK 9
//   _RetractReedsUsed: Data Word for Number of Retract Reeds used
_retractReedUsed4 := _RetractReedsUsed >= 4;

// NETWORK 10
//   _RetractReedsUsed: Data Word for Number of Retract Reeds used
//   _RetractReed1: AT %I*
//   _RetractReed2: AT %I*
//   _RetractReed3: AT %I*
//   _RetractReed4: AT %I*
//   _DualSolenoid: Configured as a dual Solenoid Device
//   _SingleSolenoidReverse: Configured as a Signal Solenoid Retract Device
//   _RetractSolOnTime_ET: Time Retract Solenoid Has Been Energised
//   _SingleSolenoidNormal: Configured as a Signal Solenoid Extend Device (Default)
//   _ExtendSolOffTime_ET: Time Since Extend Solenoid was Last Energised
//   _RetractReed: All cylinder retract reeds have been made
_RetractReed := _RetractReedsUsed > 0 AND (_RetractReed1 OR NOT _retractReedUsed1) AND (_RetractReed2 OR NOT _retractReedUsed2) AND (_RetractReed3 OR NOT _retractReedUsed3) AND (_RetractReed4 OR NOT _retractReedUsed4) OR _RetractReedsUsed = 0 AND (_DualSolenoid OR _SingleSolenoidReverse) AND _RetractSolOnTime_ET > _RtFaultTime_PT OR _RetractReedsUsed = 0 AND _SingleSolenoidNormal AND _ExtendSolOffTime_ET > _RtFaultTime_PT;
END_METHOD

METHOD PRIVATE M_ReedFault
VAR_INPUT
END_VAR
VAR_INST
	_reedFault					: BOOL;
	_reedFault_Q				: BOOL;
	_reedFaultArray				: ARRAY[0..4] OF BOOL;
END_VAR
VAR_INST // added by the converter: edge detectors and wires of the graphical bodies
    _w1, _w2, _w3, _w4, _w5 : BOOL;
END_VAR
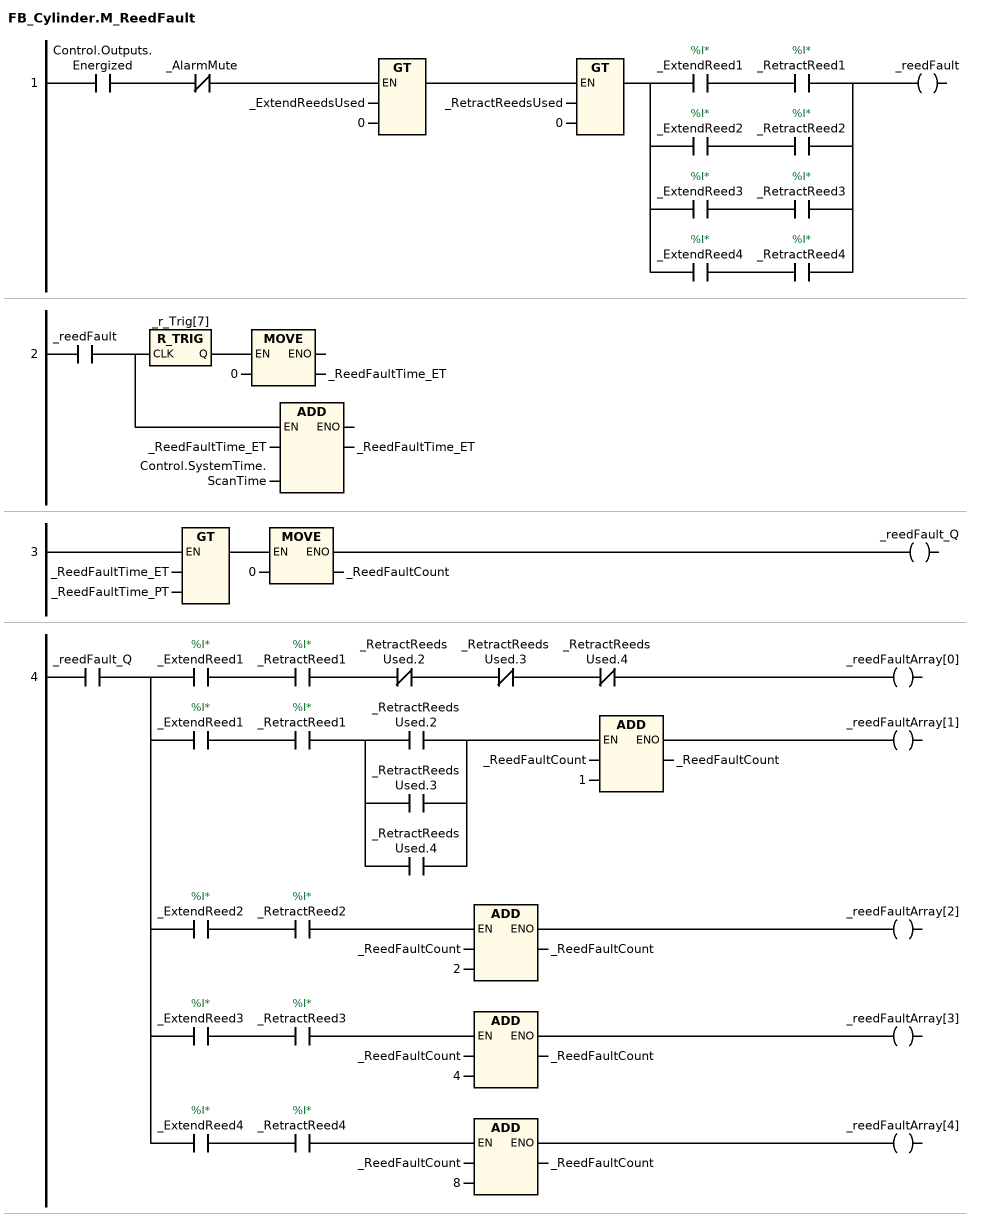
// NETWORK 1
//   _ExtendReedsUsed: Data Word for Number of Extend Reeds used
//   _RetractReedsUsed: Data Word for Number of Retract Reeds used
//   _ExtendReed1: AT %I*
//   _RetractReed1: AT %I*
//   _ExtendReed2: AT %I*
//   _RetractReed2: AT %I*
//   _ExtendReed3: AT %I*
//   _RetractReed3: AT %I*
//   _ExtendReed4: AT %I*
//   _RetractReed4: AT %I*
_reedFault := (Control.Outputs.Energized AND NOT _AlarmMute AND _ExtendReedsUsed > 0 AND _RetractReedsUsed > 0) AND (_ExtendReed1 AND _RetractReed1 OR _ExtendReed2 AND _RetractReed2 OR _ExtendReed3 AND _RetractReed3 OR _ExtendReed4 AND _RetractReed4);

// NETWORK 2
//   _ReedFaultTime_ET: Reed fault elapsed time
//   Control.SystemTime.ScanTime: Last scan time (Seconds)
_r_Trig[7](CLK := _reedFault); // R_TRIG
IF _r_Trig[7].Q THEN _ReedFaultTime_ET := 0; END_IF
IF _reedFault THEN _ReedFaultTime_ET := _ReedFaultTime_ET + Control.SystemTime.ScanTime; END_IF

// NETWORK 3
//   _ReedFaultTime_ET: Reed fault elapsed time
//   _ReedFaultCount: Count for type of reed fault
_w1 := _ReedFaultTime_ET > _ReedFaultTime_PT;
IF _w1 THEN _ReedFaultCount := 0; END_IF
_reedFault_Q := _w1;

// NETWORK 4
//   _ExtendReed1: AT %I*
//   _RetractReed1: AT %I*
//   _ReedFaultCount: Count for type of reed fault
//   _ExtendReed2: AT %I*
//   _RetractReed2: AT %I*
//   _ExtendReed3: AT %I*
//   _RetractReed3: AT %I*
//   _ExtendReed4: AT %I*
//   _RetractReed4: AT %I*
_reedFaultArray[0] := _reedFault_Q AND _ExtendReed1 AND _RetractReed1 AND NOT _RetractReedsUsed.2 AND NOT _RetractReedsUsed.3 AND NOT _RetractReedsUsed.4;
_w2 := _reedFault_Q AND _ExtendReed1 AND _RetractReed1 AND (_RetractReedsUsed.2 OR _RetractReedsUsed.3 OR _RetractReedsUsed.4);
IF _w2 THEN _ReedFaultCount := _ReedFaultCount + 1; END_IF
_reedFaultArray[1] := _w2;
_w3 := _reedFault_Q AND _ExtendReed2 AND _RetractReed2;
IF _w3 THEN _ReedFaultCount := _ReedFaultCount + 2; END_IF
_reedFaultArray[2] := _w3;
_w4 := _reedFault_Q AND _ExtendReed3 AND _RetractReed3;
IF _w4 THEN _ReedFaultCount := _ReedFaultCount + 4; END_IF
_reedFaultArray[3] := _w4;
_w5 := _reedFault_Q AND _ExtendReed4 AND _RetractReed4;
IF _w5 THEN _ReedFaultCount := _ReedFaultCount + 8; END_IF
_reedFaultArray[4] := _w5;
END_METHOD

METHOD PRIVATE M_Retract
VAR_INPUT
END_VAR
VAR_INST
END_VAR
VAR_INST // added by the converter: edge detectors and wires of the graphical bodies
    _w1, _w2 : BOOL;
END_VAR
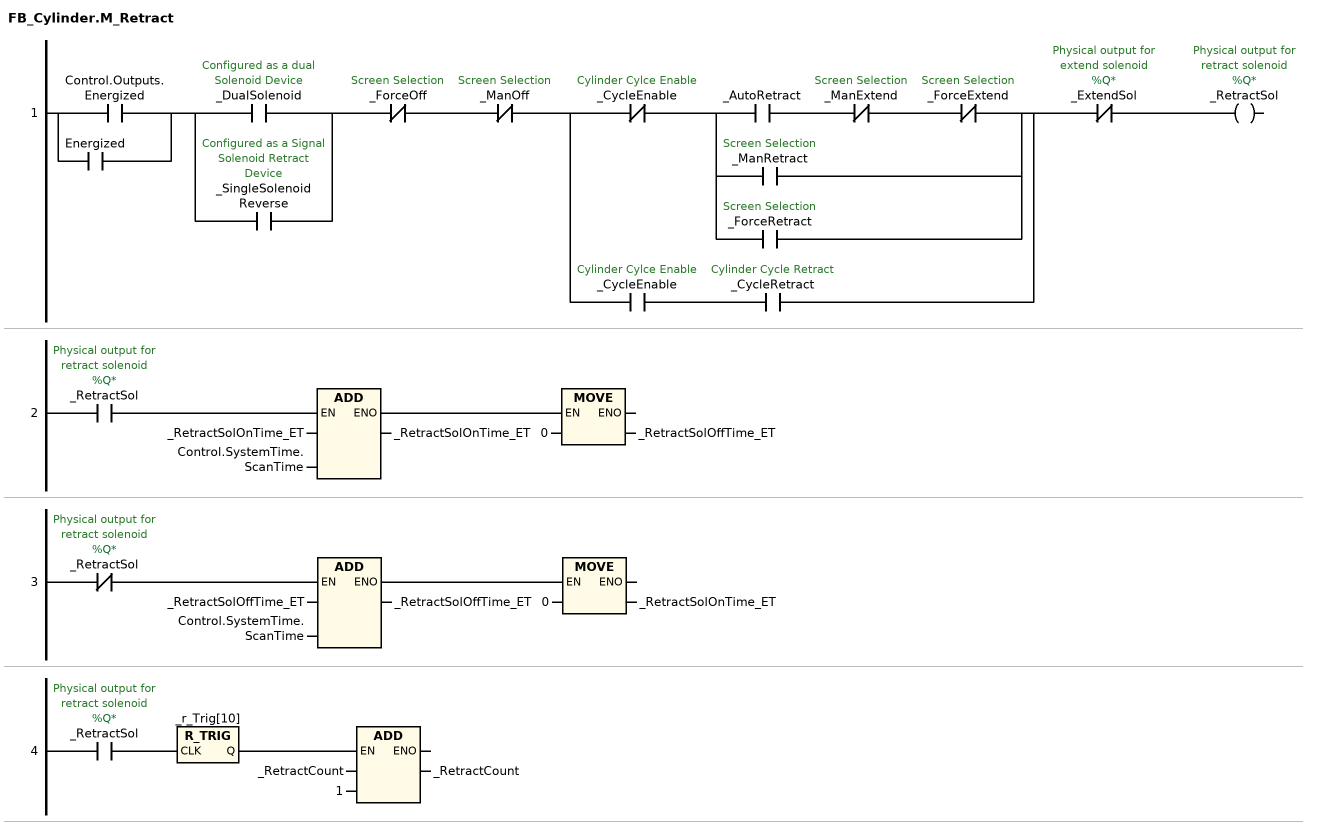
// NETWORK 1
//   _DualSolenoid: Configured as a dual Solenoid Device
//   _SingleSolenoidReverse: Configured as a Signal Solenoid Retract Device
//   _ForceOff: Screen Selection
//   _ManOff: Screen Selection
//   _CycleEnable: Cylinder Cylce Enable
//   _ManExtend: Screen Selection
//   _ForceExtend: Screen Selection
//   _ManRetract: Screen Selection
//   _ForceRetract: Screen Selection
//   _CycleRetract: Cylinder Cycle Retract
//   _ExtendSol: Physical output for extend solenoid | AT %Q*
//   _RetractSol: Physical output for retract solenoid | AT %Q*
_RetractSol := (Control.Outputs.Energized OR Energized) AND (_DualSolenoid OR _SingleSolenoidReverse) AND NOT _ForceOff AND NOT _ManOff AND (NOT _CycleEnable AND (_AutoRetract AND NOT _ManExtend AND NOT _ForceExtend OR _ManRetract OR _ForceRetract) OR _CycleEnable AND _CycleRetract) AND NOT _ExtendSol;

// NETWORK 2
//   _RetractSol: Physical output for retract solenoid | AT %Q*
//   _RetractSolOnTime_ET: Time Retract Solenoid Has Been Energised
//   Control.SystemTime.ScanTime: Last scan time (Seconds)
//   _RetractSolOffTime_ET: Time Since Retract Solenoid was Last Energised
_w1 := _RetractSol;
IF _w1 THEN _RetractSolOnTime_ET := _RetractSolOnTime_ET + Control.SystemTime.ScanTime; END_IF
IF _w1 THEN _RetractSolOffTime_ET := 0; END_IF

// NETWORK 3
//   _RetractSol: Physical output for retract solenoid | AT %Q*
//   _RetractSolOffTime_ET: Time Since Retract Solenoid was Last Energised
//   Control.SystemTime.ScanTime: Last scan time (Seconds)
//   _RetractSolOnTime_ET: Time Retract Solenoid Has Been Energised
_w2 := NOT _RetractSol;
IF _w2 THEN _RetractSolOffTime_ET := _RetractSolOffTime_ET + Control.SystemTime.ScanTime; END_IF
IF _w2 THEN _RetractSolOnTime_ET := 0; END_IF

// NETWORK 4
//   _RetractSol: Physical output for retract solenoid | AT %Q*
//   _RetractCount: Total number of cylinder retracts
_r_Trig[10](CLK := _RetractSol); // R_TRIG
IF _r_Trig[10].Q THEN _RetractCount := _RetractCount + 1; END_IF
END_METHOD

METHOD PRIVATE M_RetractFault
VAR_INPUT
END_VAR
VAR_INST
	_retracting					: BOOL;
	_retractReedFault_Q			: BOOL;
	_retractReedFaultArray		: ARRAY[0..4] OF BOOL;
END_VAR
VAR_INST // added by the converter: edge detectors and wires of the graphical bodies
    _w1, _w2, _w3, _w4, _w5 : BOOL;
END_VAR
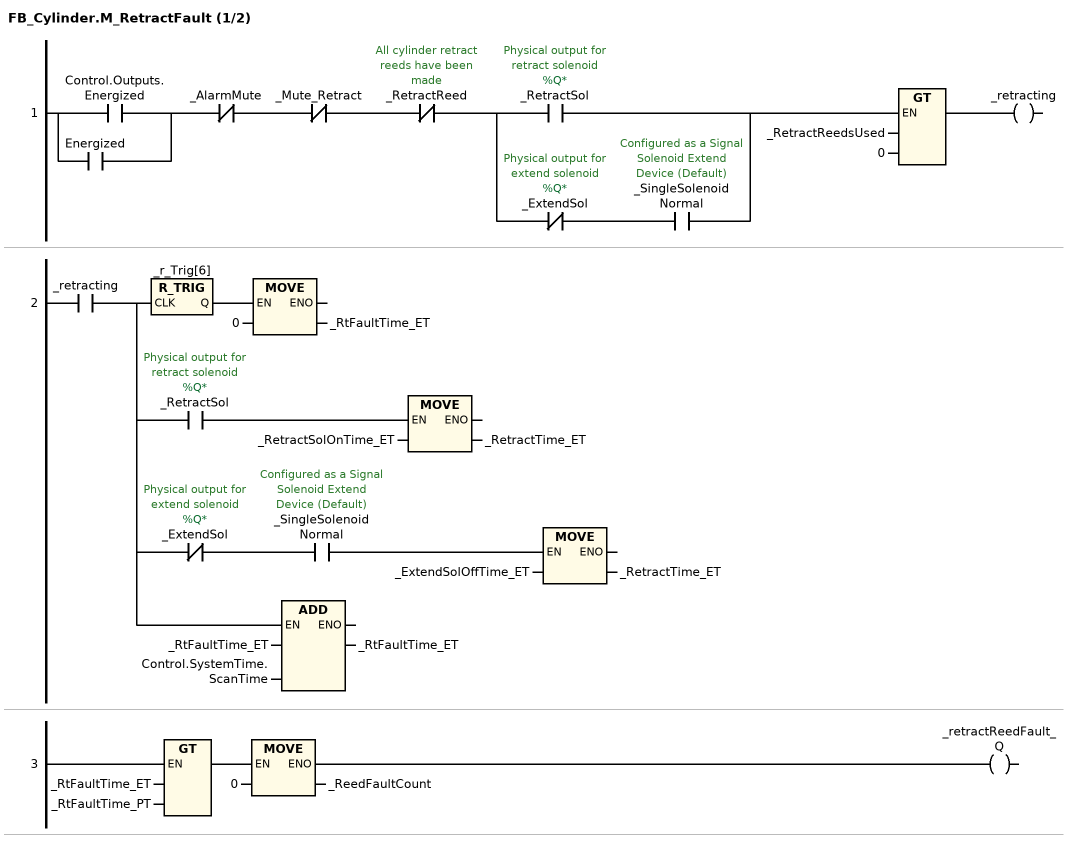
// NETWORK 1
//   _RetractReed: All cylinder retract reeds have been made
//   _RetractSol: Physical output for retract solenoid | AT %Q*
//   _ExtendSol: Physical output for extend solenoid | AT %Q*
//   _SingleSolenoidNormal: Configured as a Signal Solenoid Extend Device (Default)
//   _RetractReedsUsed: Data Word for Number of Retract Reeds used
_retracting := (Control.Outputs.Energized OR Energized) AND NOT _AlarmMute AND NOT _Mute_Retract AND NOT _RetractReed AND (_RetractSol OR NOT _ExtendSol AND _SingleSolenoidNormal) AND _RetractReedsUsed > 0;

// NETWORK 2
//   _RtFaultTime_ET: Retract fault elapsed time
//   _RetractSol: Physical output for retract solenoid | AT %Q*
//   _RetractSolOnTime_ET: Time Retract Solenoid Has Been Energised
//   _RetractTime_ET: Time Cylinder has been Retracted
//   _ExtendSol: Physical output for extend solenoid | AT %Q*
//   _SingleSolenoidNormal: Configured as a Signal Solenoid Extend Device (Default)
//   _ExtendSolOffTime_ET: Time Since Extend Solenoid was Last Energised
//   Control.SystemTime.ScanTime: Last scan time (Seconds)
_r_Trig[6](CLK := _retracting); // R_TRIG
IF _r_Trig[6].Q THEN _RtFaultTime_ET := 0; END_IF
IF _retracting AND _RetractSol THEN _RetractTime_ET := _RetractSolOnTime_ET; END_IF
IF _retracting AND NOT _ExtendSol AND _SingleSolenoidNormal THEN _RetractTime_ET := _ExtendSolOffTime_ET; END_IF
IF _retracting THEN _RtFaultTime_ET := _RtFaultTime_ET + Control.SystemTime.ScanTime; END_IF

// NETWORK 3
//   _RtFaultTime_ET: Retract fault elapsed time
//   _ReedFaultCount: Count for type of reed fault
_w1 := _RtFaultTime_ET > _RtFaultTime_PT;
IF _w1 THEN _ReedFaultCount := 0; END_IF
_retractReedFault_Q := _w1;

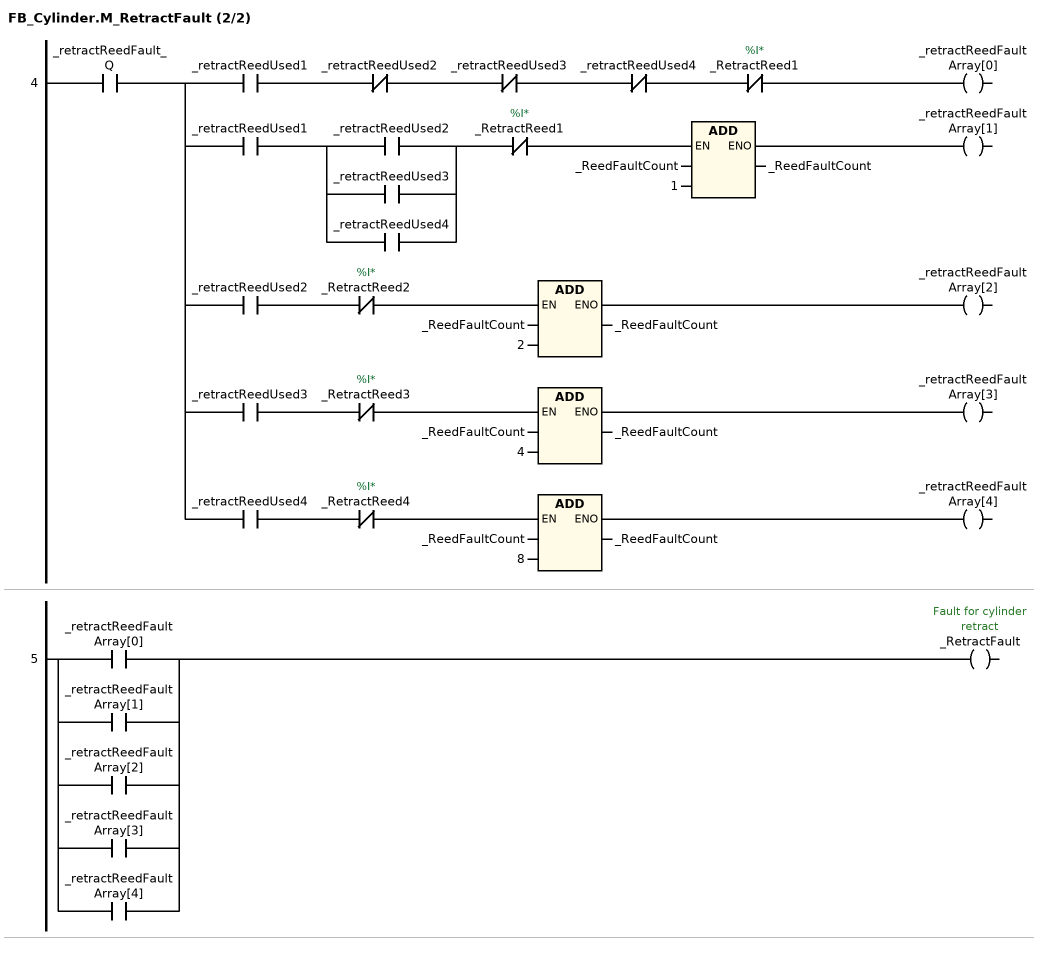
// NETWORK 4
//   _RetractReed1: AT %I*
//   _ReedFaultCount: Count for type of reed fault
//   _RetractReed2: AT %I*
//   _RetractReed3: AT %I*
//   _RetractReed4: AT %I*
_retractReedFaultArray[0] := _retractReedFault_Q AND _retractReedUsed1 AND NOT _retractReedUsed2 AND NOT _retractReedUsed3 AND NOT _retractReedUsed4 AND NOT _RetractReed1;
_w2 := _retractReedFault_Q AND _retractReedUsed1 AND (_retractReedUsed2 OR _retractReedUsed3 OR _retractReedUsed4) AND NOT _RetractReed1;
IF _w2 THEN _ReedFaultCount := _ReedFaultCount + 1; END_IF
_retractReedFaultArray[1] := _w2;
_w3 := _retractReedFault_Q AND _retractReedUsed2 AND NOT _RetractReed2;
IF _w3 THEN _ReedFaultCount := _ReedFaultCount + 2; END_IF
_retractReedFaultArray[2] := _w3;
_w4 := _retractReedFault_Q AND _retractReedUsed3 AND NOT _RetractReed3;
IF _w4 THEN _ReedFaultCount := _ReedFaultCount + 4; END_IF
_retractReedFaultArray[3] := _w4;
_w5 := _retractReedFault_Q AND _retractReedUsed4 AND NOT _RetractReed4;
IF _w5 THEN _ReedFaultCount := _ReedFaultCount + 8; END_IF
_retractReedFaultArray[4] := _w5;

// NETWORK 5
//   _RetractFault: Fault for cylinder retract
_RetractFault := _retractReedFaultArray[0] OR _retractReedFaultArray[1] OR _retractReedFaultArray[2] OR _retractReedFaultArray[3] OR _retractReedFaultArray[4];
END_METHOD

METHOD PRIVATE M_TestCycle
VAR_INPUT
END_VAR
VAR_INST
END_VAR
VAR_INST // added by the converter: edge detectors and wires of the graphical bodies
    _w1, _w2, _w3 : BOOL;
END_VAR
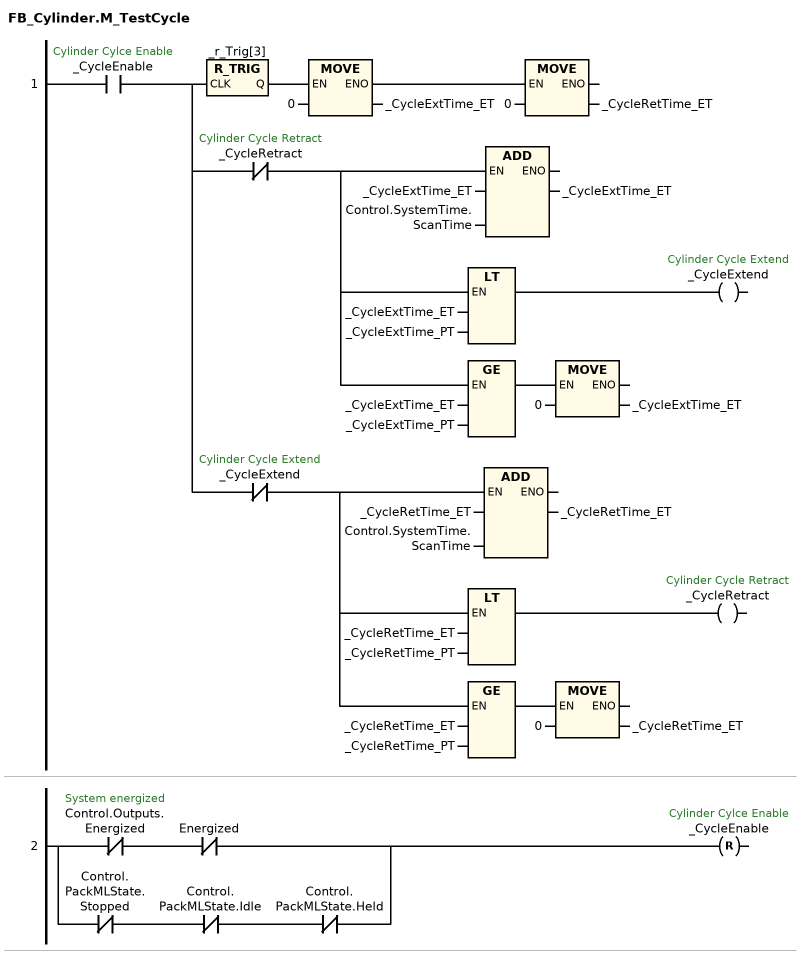
// NETWORK 1
//   _CycleEnable: Cylinder Cylce Enable
//   _CycleExtTime_ET: Cylinder Cycle Extend Accumulated Time
//   _CycleRetTime_ET: Cylinder Cycle Retract Accumulated Time
//   _CycleRetract: Cylinder Cycle Retract
//   Control.SystemTime.ScanTime: Last scan time (Seconds)
//   _CycleExtTime_PT: Cylinder Cycle Extend Time Preset
//   _CycleExtend: Cylinder Cycle Extend
//   _CycleRetTime_PT: Cylinder Cycle Retract Time Preset
_r_Trig[3](CLK := _CycleEnable); // R_TRIG
_w1 := _r_Trig[3].Q;
IF _w1 THEN _CycleExtTime_ET := 0; END_IF
IF _w1 THEN _CycleRetTime_ET := 0; END_IF
_w2 := _CycleEnable AND NOT _CycleRetract;
IF _w2 THEN _CycleExtTime_ET := _CycleExtTime_ET + Control.SystemTime.ScanTime; END_IF
_CycleExtend := _w2 AND _CycleExtTime_ET < _CycleExtTime_PT;
IF _w2 AND _CycleExtTime_ET >= _CycleExtTime_PT THEN _CycleExtTime_ET := 0; END_IF
_w3 := _CycleEnable AND NOT _CycleExtend;
IF _w3 THEN _CycleRetTime_ET := _CycleRetTime_ET + Control.SystemTime.ScanTime; END_IF
_CycleRetract := _w3 AND _CycleRetTime_ET < _CycleRetTime_PT;
IF _w3 AND _CycleRetTime_ET >= _CycleRetTime_PT THEN _CycleRetTime_ET := 0; END_IF

// NETWORK 2
//   Control.Outputs.Energized: System energized
//   _CycleEnable: Cylinder Cylce Enable
_CycleEnable R= NOT Control.Outputs.Energized AND NOT Energized OR NOT Control.PackMLState.Stopped AND NOT Control.PackMLState.Idle AND NOT Control.PackMLState.Held;
END_METHOD

METHOD PRIVATE M_TypeConfig
VAR_INPUT
END_VAR
VAR_INST
END_VAR
CASE _TypeCfg OF
	eCylinderType_SINGLE_NORMAL : 
		_SingleSolenoidNormal := TRUE;
		_SingleSolenoidReverse := FALSE;
		_DualSolenoid := FALSE;
	eCylinderType_SINGLE_REVERSE : 
		_SingleSolenoidNormal := FALSE;
		_SingleSolenoidReverse := TRUE;
		_DualSolenoid := FALSE;
	eCylinderType_DUEL : 
		_SingleSolenoidNormal := FALSE;
		_SingleSolenoidReverse := FALSE;
		_DualSolenoid := TRUE;
END_CASE
END_METHOD

METHOD PRIVATE M_UnlatchManuals
VAR_INPUT
END_VAR
VAR_INST // added by the converter: edge detectors and wires of the graphical bodies
    _rt1, _rt2, _rt3, _rt4 : R_TRIG;
END_VAR
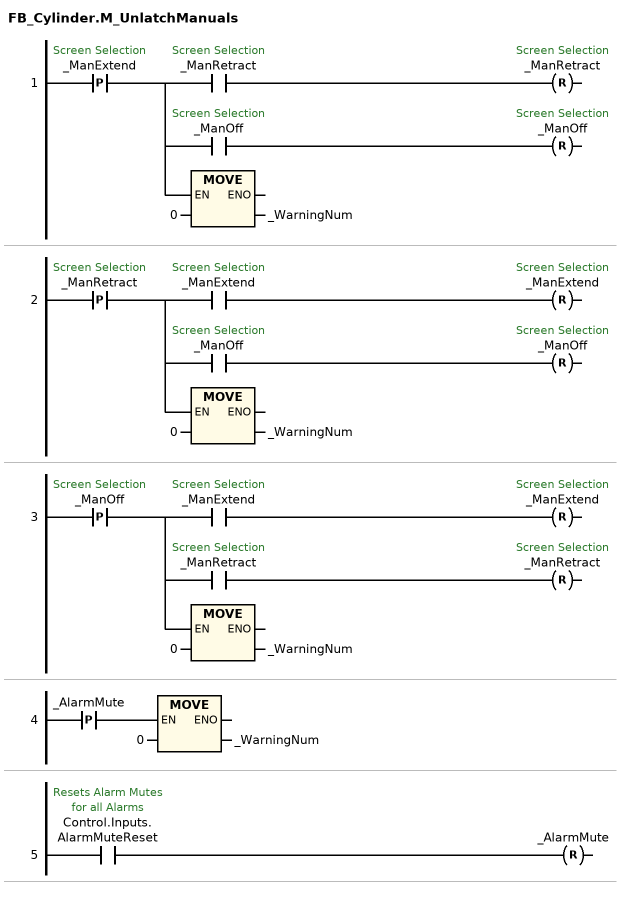
// NETWORK 1
//   _ManExtend: Screen Selection
//   _ManRetract: Screen Selection
//   _ManOff: Screen Selection
_rt1(CLK := _ManExtend);
_ManRetract R= _rt1.Q AND _ManRetract;
_ManOff R= _rt1.Q AND _ManOff;
IF _rt1.Q THEN _WarningNum := 0; END_IF

// NETWORK 2
//   _ManRetract: Screen Selection
//   _ManExtend: Screen Selection
//   _ManOff: Screen Selection
_rt2(CLK := _ManRetract);
_ManExtend R= _rt2.Q AND _ManExtend;
_ManOff R= _rt2.Q AND _ManOff;
IF _rt2.Q THEN _WarningNum := 0; END_IF

// NETWORK 3
//   _ManOff: Screen Selection
//   _ManExtend: Screen Selection
//   _ManRetract: Screen Selection
_rt3(CLK := _ManOff);
_ManExtend R= _rt3.Q AND _ManExtend;
_ManRetract R= _rt3.Q AND _ManRetract;
IF _rt3.Q THEN _WarningNum := 0; END_IF

// NETWORK 4
_rt4(CLK := _AlarmMute);
IF _rt4.Q THEN _WarningNum := 0; END_IF

// NETWORK 5
//   Control.Inputs.AlarmMuteReset: Resets Alarm Mutes for all Alarms
_AlarmMute R= Control.Inputs.AlarmMuteReset;
END_METHOD

METHOD PRIVATE M_WarningMonitor
VAR_INPUT
END_VAR
VAR_INST // added by the converter: edge detectors and wires of the graphical bodies
    _w1, _w2, _w3, _w4, _w5, _w6, _w7 : BOOL;
END_VAR
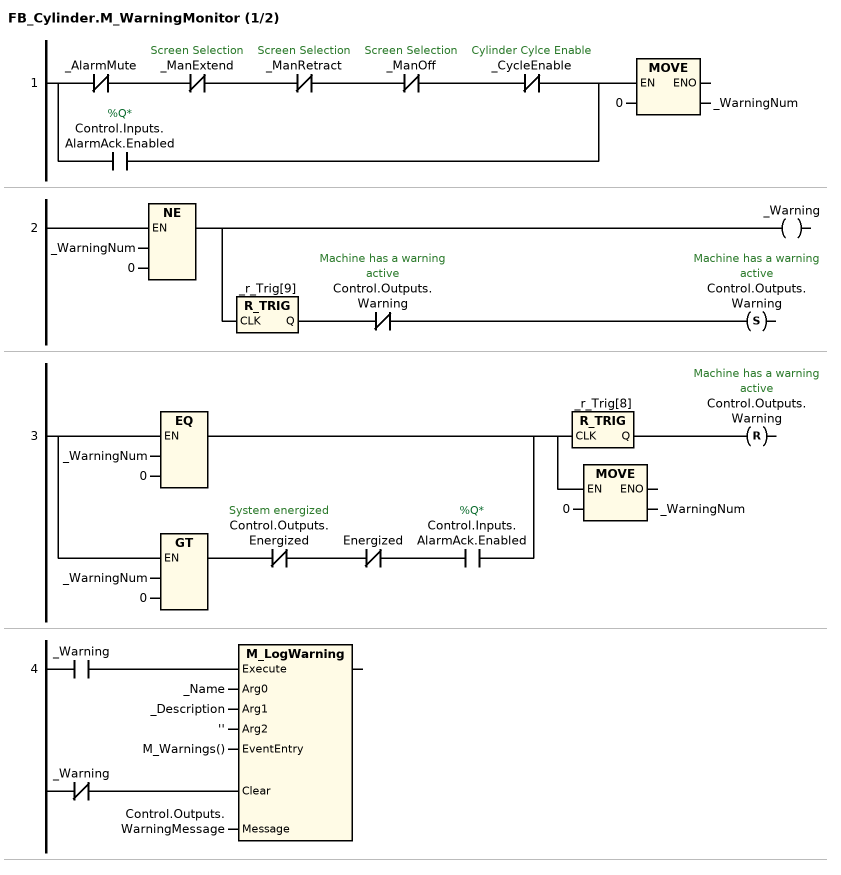
// NETWORK 1
//   _ManExtend: Screen Selection
//   _ManRetract: Screen Selection
//   _ManOff: Screen Selection
//   _CycleEnable: Cylinder Cylce Enable
//   Control.Inputs.AlarmAck.Enabled: AT %Q*
IF NOT _AlarmMute AND NOT _ManExtend AND NOT _ManRetract AND NOT _ManOff AND NOT _CycleEnable OR Control.Inputs.AlarmAck.Enabled THEN
    _WarningNum := 0;
END_IF

// NETWORK 2
//   Control.Outputs.Warning: Machine has a warning active
_w1 := _WarningNum <> 0;
_Warning := _w1;
_r_Trig[9](CLK := _w1); // R_TRIG
Control.Outputs.Warning S= _r_Trig[9].Q AND NOT Control.Outputs.Warning;

// NETWORK 3
//   Control.Outputs.Energized: System energized
//   Control.Inputs.AlarmAck.Enabled: AT %Q*
//   Control.Outputs.Warning: Machine has a warning active
_w2 := _WarningNum = 0 OR _WarningNum > 0 AND NOT Control.Outputs.Energized AND NOT Energized AND Control.Inputs.AlarmAck.Enabled;
_r_Trig[8](CLK := _w2); // R_TRIG
Control.Outputs.Warning R= _r_Trig[8].Q;
IF _w2 THEN _WarningNum := 0; END_IF

// NETWORK 4
M_LogWarning(Execute := _Warning, Arg0 := _Name, Arg1 := _Description, Arg2 := '', EventEntry := M_Warnings(), Clear := NOT _Warning, Message := Control.Outputs.WarningMessage);

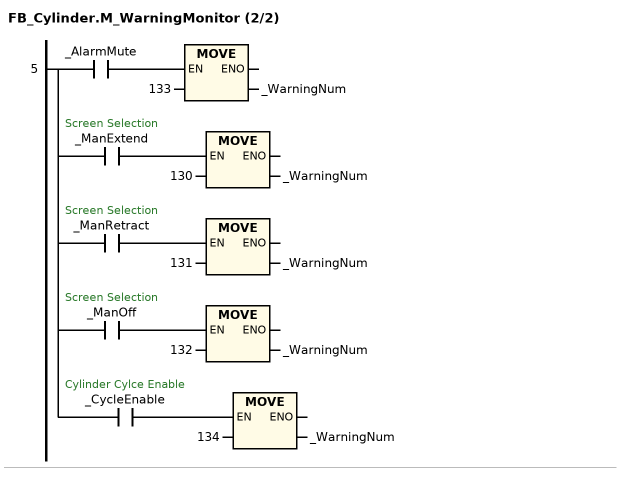
// NETWORK 5
//   _ManExtend: Screen Selection
//   _ManRetract: Screen Selection
//   _ManOff: Screen Selection
//   _CycleEnable: Cylinder Cylce Enable
_w3 := _AlarmMute;
IF _w3 THEN _WarningNum := 133; END_IF
_w4 := _ManExtend;
IF _w4 THEN _WarningNum := 130; END_IF
_w5 := _ManRetract;
IF _w5 THEN _WarningNum := 131; END_IF
_w6 := _ManOff;
IF _w6 THEN _WarningNum := 132; END_IF
_w7 := _CycleEnable;
IF _w7 THEN _WarningNum := 134; END_IF
(* _w3 OR _w4 OR _w5 OR _w6 OR _w7; result not used *)
END_METHOD

METHOD PRIVATE M_Warnings : TcEventEntry
VAR_INPUT
END_VAR
CASE _WarningNum OF
	130: M_Warnings:= TC_Events.TcCylinder.W_130;//Manual Extend Enabled	
	131: M_Warnings:= TC_Events.TcCylinder.W_131;//Manual Retract Enabled		
	132: M_Warnings:= TC_Events.TcCylinder.W_132;//Manual OFF Enabled
	133: M_Warnings:= TC_Events.TcCylinder.W_133;//Alarm Mute Active
	134: M_Warnings:= TC_Events.TcCylinder.W_134;//Cylinder Cycling Enabled					
ELSE
	M_Warnings:=  TC_Events.TcCylinder.W_Undefined;
END_CASE
END_METHOD

{attribute 'monitoring' := 'variable'}
PROPERTY PUBLIC ManExtend : Bool
GET
ManExtend := _ManExtend;
END_GET
SET
_ManExtend := ManExtend;
END_SET
END_PROPERTY

{attribute 'monitoring' := 'variable'}
PROPERTY PUBLIC ManOff : Bool
GET
ManOff := _ManOff;
END_GET
SET
_ManOff := ManOff;
END_SET
END_PROPERTY

{attribute 'monitoring' := 'variable'}
PROPERTY PUBLIC ManRetract : Bool
GET
ManRetract := _ManRetract;
END_GET
SET
_ManRetract := ManRetract;
END_SET
END_PROPERTY

{attribute 'monitoring' := 'variable'}
PROPERTY PUBLIC Name : String[15]
GET
Name := _Name;
END_GET
SET
_Name := Name;
END_SET
END_PROPERTY

{attribute 'monitoring' := 'variable'}
PROPERTY PUBLIC ReedFaultTime_ET : real
GET
ReedFaultTime_ET := _ReedFaultTime_ET;
END_GET
END_PROPERTY

{attribute 'monitoring' := 'variable'}
PROPERTY PUBLIC ReedFaultTime_PT : real
GET
ReedFaultTime_PT := _ReedFaultTime_PT;
END_GET
SET
_ReedFaultTime_PT := ReedFaultTime_PT;
END_SET
END_PROPERTY

{attribute 'monitoring' := 'variable'}
PROPERTY PUBLIC RetractReed : Bool
GET
RetractReed := _RetractReed;
END_GET
END_PROPERTY

{attribute 'monitoring' := 'variable'}
PROPERTY PUBLIC RetractReed1 : Bool
GET
RetractReed1 := _RetractReed1;
END_GET
SET
PUBLIC 
VAR
END_VAR
_RetractReed1 := RetractReed1;
END_SET
END_PROPERTY

{attribute 'monitoring' := 'variable'}
PROPERTY PUBLIC RetractSol : Bool
GET
RetractSol := _RetractSol;
END_GET
END_PROPERTY

{attribute 'monitoring' := 'variable'}
PROPERTY PUBLIC RtFaultTime_ET : real
GET
RtFaultTime_ET := _RtFaultTime_ET;
END_GET
END_PROPERTY

{attribute 'monitoring' := 'variable'}
PROPERTY PUBLIC RtFaultTime_PT : real
GET
RtFaultTime_PT := _RtFaultTime_PT;
END_GET
SET
_RtFaultTime_PT := RtFaultTime_PT;
END_SET
END_PROPERTY

{attribute 'monitoring' := 'variable'}
PROPERTY PUBLIC StandbyReset : Bool
GET
StandbyReset := _ForceOff;
END_GET
SET
_ForceOff := StandbyReset;
END_SET
END_PROPERTY

PROPERTY PUBLIC Variables : REFERENCE TO ARRAY[0..9] OF ST_Variable
GET
Variables REF= _Variables;
END_GET
END_PROPERTY

{attribute 'monitoring' := 'variable'}
PROPERTY PUBLIC Warning : Bool
GET
Warning := _Warning;
END_GET
END_PROPERTY

END_FUNCTION_BLOCK

// Objects/FB_Database_V4_00/Stored Procedures/FB_Example
FUNCTION_BLOCK FB_Example EXTENDS FB_Tc2Database 
VAR_INPUT
	Execute					: BOOL;//Execute Stored Procedure
	TimeStamp				: DT;//Current Time
	Uid						: STRING(31);//8 Byte Unique Mac Id
	DataOk					: USINT;//0=Fail, 1=Pass, 2=NA
	VisionOk				: USINT;//0=Fail, 1=Pass, 2=NA
	VisionCause				: USINT;//Cause of Vision Failure if Applicable	
	VisionScore				: USINT;//0-100% Tag Find Score	
	GetCycles				: BOOL;//Get Tag Cycle Anount
	GetAge					: BOOL;//Get Tag Age
	GetRecord				: BOOL;//Get Record History
	Expired					: BOOL;//Tag Expired
END_VAR
VAR_IN_OUT         
	Record					: ARRAY[0..29] OF ST_Example;
END_VAR
VAR_OUTPUT
	Busy					: BOOL;
END_VAR
VAR
	_State					: UINT;
	_fb_SPRecordArray		: FB_DBStoredProceduresRecordArray;
	_ParameterList			: ARRAY[0..9] OF ST_DBParameter;
END_VAR

Name :=  'Insert';
Description:= 'FB_Example';

_fb_SPRecordArray(
	sNetID:= '', 
	hDBID:= 1, 
	sProcedureName:= 'USP_Example',
	cbParameterList:= SIZEOF(_ParameterList),
	pParameterList:= ADR(_ParameterList),
	nStartIndex:= 0, 
	nRecordCount:= SIZEOF(Record)/SIZEOF(Record[0]), 
	bExecute:= , 
	tTimeout:= T#10S, 
	pDestAddr:=  ADR(Record),
	cbRecordArraySize:= SIZEOF(Record), 
	bBusy=> Busy, 
	bError=> , 
	nErrID=> , 
	sSQLState=> , 
	nRecords=> );

CASE _State OF	
0:	
	IF Execute AND NOT Busy THEN
		_State:= 1;
	END_IF
1:
	_ParameterList[0].sParameterName := '@TimeStamped';
	_ParameterList[0].eParameterDataType := eDBColumn_DateTime;
	_ParameterList[0].eParameterType := eDBParameter_Input;
	_ParameterList[0].cbParameterValue := SIZEOF(TimeStamp);
	_ParameterList[0].pParameterValue := ADR(TimeStamp);
	
	_ParameterList[1].sParameterName := '@Uid';
	_ParameterList[1].eParameterDataType := eDBColumn_NVarChar;
	_ParameterList[1].eParameterType := eDBParameter_Input;
	_ParameterList[1].cbParameterValue := SIZEOF(Uid);
	_ParameterList[1].pParameterValue := ADR(Uid);
	
	_ParameterList[2].sParameterName := '@DataOk';
	_ParameterList[2].eParameterDataType := eDBColumn_TinyInt;
	_ParameterList[2].eParameterType := eDBParameter_Input;
	_ParameterList[2].cbParameterValue := SIZEOF(DataOk);
	_ParameterList[2].pParameterValue := ADR(DataOk);
	
	_ParameterList[3].sParameterName := '@VisionOk';
	_ParameterList[3].eParameterDataType := eDBColumn_TinyInt;
	_ParameterList[3].eParameterType := eDBParameter_Input;
	_ParameterList[3].cbParameterValue := SIZEOF(VisionOk);
	_ParameterList[3].pParameterValue := ADR(VisionOk);
	
	_ParameterList[4].sParameterName := '@VisionCause';
	_ParameterList[4].eParameterDataType := eDBColumn_TinyInt;
	_ParameterList[4].eParameterType := eDBParameter_Input;
	_ParameterList[4].cbParameterValue := SIZEOF(VisionCause);
	_ParameterList[4].pParameterValue := ADR(VisionCause);
	
	_ParameterList[5].sParameterName := '@VisionScore';
	_ParameterList[5].eParameterDataType := eDBColumn_TinyInt;
	_ParameterList[5].eParameterType := eDBParameter_Input;
	_ParameterList[5].cbParameterValue := SIZEOF(VisionScore);
	_ParameterList[5].pParameterValue := ADR(VisionScore);
	
	_ParameterList[6].sParameterName := '@GetCycles';
	_ParameterList[6].eParameterDataType := eDBColumn_Bit;
	_ParameterList[6].eParameterType := eDBParameter_Input;
	_ParameterList[6].cbParameterValue := SIZEOF(GetCycles);
	_ParameterList[6].pParameterValue := ADR(GetCycles);
	
	_ParameterList[7].sParameterName := '@GetAge';
	_ParameterList[7].eParameterDataType := eDBColumn_Bit;
	_ParameterList[7].eParameterType := eDBParameter_Input;
	_ParameterList[7].cbParameterValue := SIZEOF(GetAge);
	_ParameterList[7].pParameterValue := ADR(GetAge);
	
	_ParameterList[8].sParameterName := '@GetRecord';
	_ParameterList[8].eParameterDataType := eDBColumn_Bit;
	_ParameterList[8].eParameterType := eDBParameter_Input;
	_ParameterList[8].cbParameterValue := SIZEOF(GetRecord);
	_ParameterList[8].pParameterValue := ADR(GetRecord);
	
	_ParameterList[9].sParameterName := '@Expired';
	_ParameterList[9].eParameterDataType := eDBColumn_Bit;
	_ParameterList[9].eParameterType := eDBParameter_Input;
	_ParameterList[9].cbParameterValue := SIZEOF(Expired);
	_ParameterList[9].pParameterValue := ADR(Expired);
	_State:= 2;
	
2:
	_fb_SPRecordArray.bExecute := TRUE;
	_State:= 3;
3:
	IF NOT Execute THEN
		_fb_SPRecordArray.bExecute := FALSE;
		_State:= 0;
	END_IF
	
END_CASE

M_AlarmMonitor(Error:= _fb_SPRecordArray.bError, ErrorID:= _fb_SPRecordArray.nErrID, DBSQLError:= _fb_SPRecordArray.sSQLState);

END_FUNCTION_BLOCK

// Objects/FB_Database_V4_00/FB_Tc2Database
FUNCTION_BLOCK FB_Tc2Database
VAR_INPUT
	DatabaseType			: E_DatabaseType;
END_VAR
VAR_IN_OUT 
	Control					: ST_System;         
END_VAR
VAR           
	_Alarm					: BOOL;						//Device Alarm
END_VAR
VAR PERSISTENT
	_Name					: STRING[15];		//Name for HMI
	_Description			: STRING[40];		//Description for HMI
	_AlarmMute				: BOOL;				//Alarm Mute
END_VAR

{attribute 'monitoring' := 'variable'}
PROPERTY PUBLIC Alarm : Bool
GET
Alarm := _Alarm;
END_GET
END_PROPERTY

{attribute 'monitoring' := 'variable'}
PROPERTY PUBLIC AlarmMute : BOOL
SET
AlarmMute := _AlarmMute;
END_SET
END_PROPERTY

{attribute 'monitoring' := 'variable'}
PROPERTY PUBLIC Description : String[40]
GET
Description := _Description;
END_GET
SET
_Description := Description;
END_SET
END_PROPERTY

METHOD PROTECTED M_AlarmMonitor
VAR_INPUT
	Error 		: BOOL;
	ErrorID		: UDINT;
	DBSQLError 	: ST_DBSQLError;
END_VAR
VAR_INST
	DbEvent 	: ARRAY[1601..1603] OF FB_SystemEvent;
END_VAR
VAR_INST // added by the converter: edge detectors and wires of the graphical bodies
    _rt1 : R_TRIG;
    _w1 : BOOL;
END_VAR
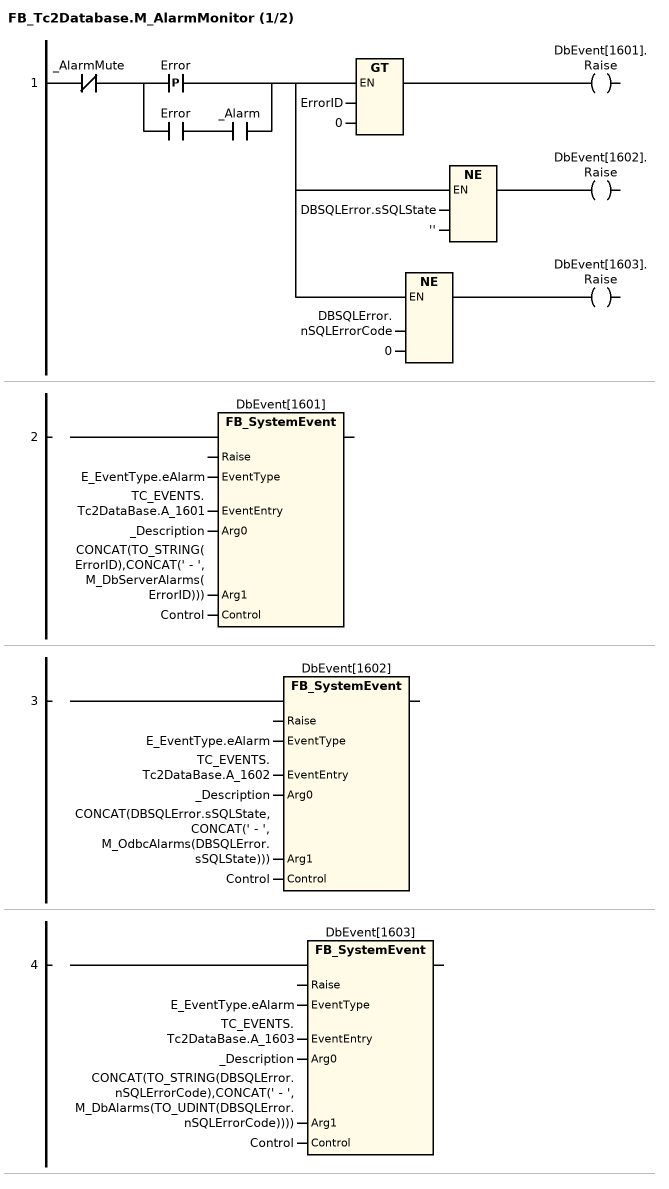
// NETWORK 1
_rt1(CLK := Error);
_w1 := NOT _AlarmMute AND (_rt1.Q OR Error AND _Alarm);
DbEvent[1601].Raise := _w1 AND ErrorID > 0;
DbEvent[1602].Raise := _w1 AND DBSQLError.sSQLState <> '';
DbEvent[1603].Raise := _w1 AND DBSQLError.nSQLErrorCode <> 0;

// NETWORK 2
DbEvent[1601](
    EventType := E_EventType.eAlarm,
    EventEntry := TC_EVENTS.Tc2DataBase.A_1601,
    Arg0 := _Description,
    Arg1 := CONCAT(TO_STRING(ErrorID),CONCAT(' - ', M_DbServerAlarms(ErrorID))),
    Control := Control); // FB_SystemEvent

// NETWORK 3
DbEvent[1602](
    EventType := E_EventType.eAlarm,
    EventEntry := TC_EVENTS.Tc2DataBase.A_1602,
    Arg0 := _Description,
    Arg1 := CONCAT(DBSQLError.sSQLState, CONCAT(' - ', M_OdbcAlarms(DBSQLError.sSQLState))),
    Control := Control); // FB_SystemEvent

// NETWORK 4
DbEvent[1603](
    EventType := E_EventType.eAlarm,
    EventEntry := TC_EVENTS.Tc2DataBase.A_1603,
    Arg0 := _Description,
    Arg1 := CONCAT(TO_STRING(DBSQLError.nSQLErrorCode),CONCAT(' - ', M_DbAlarms(TO_UDINT(DBSQLError.nSQLErrorCode)))),
    Control := Control); // FB_SystemEvent

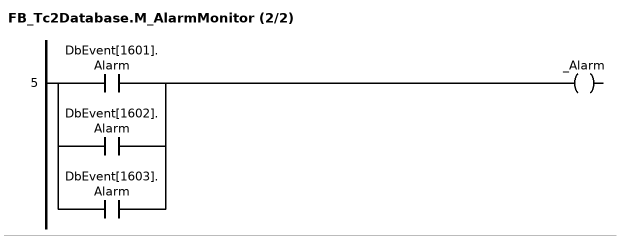
// NETWORK 5
_Alarm := DbEvent[1601].Alarm OR DbEvent[1602].Alarm OR DbEvent[1603].Alarm;
END_METHOD

